C09016=1035.593,55.483,-90.705,169.074,40.767,157.648
C09017=1035.600,55.731,-90.722,169.076,40.767,157.648
C09018=1035.606,55.981,-90.739,169.078,40.766,157.648
C09019=1035.612,56.230,-90.757,169.080,40.766,157.648
C09020=1035.619,56.479,-90.774,169.082,40.766,157.648
C09021=1035.626,56.729,-90.792,169.085,40.766,157.648
C09022=1035.631,56.978,-90.809,169.087,40.765,157.648
C09023=1035.638,57.227,-90.826,169.089,40.765,157.648
C09024=1035.645,57.477,-90.844,169.091,40.764,157.648
C09025=1035.650,57.726,-90.861,169.093,40.764,157.649
C09026=1035.657,57.976,-90.878,169.095,40.764,157.649
C09027=1035.663,58.224,-90.895,169.097,40.764,157.649
C09028=1035.669,58.474,-90.913,169.100,40.763,157.649
C09029=1035.676,58.724,-90.930,169.102,40.763,157.649
C09030=1035.682,58.973,-90.948,169.104,40.762,157.649
C09031=1035.689,59.222,-90.965,169.106,40.762,157.649
C09032=1035.695,59.471,-90.983,169.108,40.762,157.649
C09033=1035.701,59.720,-91.000,169.110,40.762,157.649
C09034=1035.708,59.970,-91.017,169.113,40.761,157.649
C09035=1035.715,60.257,-91.038,169.115,40.760,157.649
C09036=1035.722,60.543,-91.058,169.117,40.760,157.649
C09037=1035.730,60.827,-91.078,169.120,40.760,157.649
C09038=1035.738,61.114,-91.098,169.122,40.760,157.649
C09039=1035.743,61.363,-91.116,169.125,40.759,157.649
C09040=1035.750,61.613,-91.133,169.127,40.759,157.649
C09041=1035.757,61.862,-91.150,169.129,40.758,157.649
C09042=1035.763,62.112,-91.168,169.131,40.758,157.649
C09043=1035.769,62.361,-91.185,169.133,40.758,157.649
C09044=1035.776,62.610,-91.203,169.135,40.758,157.649
C09045=1035.782,62.860,-91.220,169.138,40.757,157.649
C09046=1035.789,63.109,-91.238,169.140,40.756,157.649
C09047=1035.795,63.358,-91.255,169.142,40.756,157.649
C09048=1035.802,63.608,-91.273,169.144,40.756,157.649
C09049=1035.808,63.857,-91.291,169.146,40.756,157.649
C09050=1035.814,64.105,-91.308,169.148,40.755,157.650
C09051=1035.820,64.355,-91.326,169.150,40.755,157.650
C09052=1035.827,64.605,-91.344,169.152,40.755,157.650
C09053=1035.833,64.854,-91.362,169.155,40.755,157.650
C09054=1035.839,65.103,-91.380,169.157,40.754,157.650
C09055=1035.846,65.352,-91.397,169.159,40.754,157.650
C09056=1035.852,65.602,-91.415,169.161,40.754,157.650
C09057=1035.858,65.851,-91.433,169.163,40.753,157.650
C09058=1035.865,66.100,-91.451,169.165,40.753,157.650
C09059=1035.871,66.350,-91.469,169.167,40.753,157.650
C09060=1035.877,66.599,-91.487,169.169,40.752,157.650
C09061=1035.883,66.848,-91.504,169.172,40.752,157.650
C09062=1035.890,67.097,-91.522,169.174,40.752,157.650
C09063=1035.896,67.347,-91.540,169.176,40.752,157.650
C09064=1035.903,67.596,-91.557,169.178,40.751,157.650
C09065=1035.909,67.845,-91.576,169.180,40.751,157.650
C09066=1035.915,68.094,-91.594,169.182,40.751,157.650
C09067=1035.921,68.344,-91.612,169.184,40.751,157.650
C09068=1035.928,68.593,-91.630,169.186,40.751,157.650
C09069=1035.934,68.842,-91.647,169.188,40.750,157.651
C09070=1035.940,69.092,-91.665,169.192,40.750,157.651
C09071=1035.946,69.341,-91.684,169.194,40.750,157.651
C09072=1035.953,69.590,-91.701,169.196,40.750,157.651
C09073=1035.959,69.839,-91.720,169.198,40.749,157.651
C09074=1035.965,70.088,-91.737,169.200,40.749,157.651
C09075=1035.971,70.338,-91.755,169.202,40.749,157.651
C09076=1035.978,70.587,-91.774,169.204,40.749,157.651
C09077=1035.984,70.837,-91.792,169.206,40.748,157.651
C09078=1035.990,71.085,-91.810,169.208,40.748,157.651
C09079=1035.996,71.335,-91.828,169.211,40.748,157.651
C09080=1036.003,71.584,-91.846,169.213,40.748,157.651
C09081=1036.009,71.834,-91.864,169.215,40.747,157.651
C09082=1036.015,72.083,-91.883,169.217,40.747,157.651
C09083=1036.021,72.332,-91.900,169.219,40.747,157.651
C09084=1036.027,72.581,-91.919,169.221,40.747,157.651
C09085=1036.034,72.831,-91.936,169.223,40.747,157.651
C09086=1036.041,73.080,-91.955,169.225,40.746,157.652
C09087=1036.047,73.329,-91.973,169.227,40.746,157.652
C09088=1036.053,73.579,-91.992,169.229,40.746,157.652
C09089=1036.059,73.828,-92.009,169.232,40.746,157.652
C09090=1036.065,74.077,-92.028,169.234,40.745,157.652
C09091=1036.071,74.326,-92.046,169.236,40.745,157.652
C09092=1036.078,74.576,-92.064,169.238,40.745,157.652
C09093=1036.084,74.825,-92.082,169.240,40.745,157.652
C09094=1036.091,75.074,-92.100,169.242,40.744,157.652
C09095=1036.096,75.323,-92.118,169.244,40.744,157.652
C09096=1036.103,75.572,-92.137,169.246,40.744,157.652
C09097=1036.109,75.821,-92.155,169.248,40.744,157.652
C09098=1036.115,76.071,-92.173,169.251,40.743,157.652
C09099=1036.123,76.357,-92.194,169.253,40.743,157.652
C09100=1036.130,76.643,-92.215,169.255,40.743,157.652
C09101=1036.138,76.929,-92.236,169.258,40.743,157.652
C09102=1036.144,77.215,-92.257,169.260,40.742,157.653
C09103=1036.150,77.464,-92.276,169.262,40.742,157.653
C09104=1036.157,77.713,-92.294,169.264,40.742,157.653
C09105=1036.163,77.962,-92.313,169.267,40.742,157.653
C09106=1036.169,78.212,-92.331,169.269,40.741,157.653
C09107=1036.176,78.461,-92.350,169.271,40.741,157.653
C09108=1036.182,78.710,-92.368,169.273,40.741,157.653
C09109=1036.188,78.959,-92.386,169.275,40.741,157.653
C09110=1036.194,79.209,-92.404,169.278,40.741,157.653
C09111=1036.200,79.458,-92.424,169.280,40.740,157.653
C09112=1036.206,79.707,-92.442,169.282,40.740,157.653
C09113=1036.212,79.957,-92.460,169.284,40.740,157.653
C09114=1036.219,80.206,-92.479,169.286,40.740,157.653
C09115=1036.225,80.455,-92.498,169.288,40.740,157.653
C09116=1036.232,80.704,-92.516,169.290,40.740,157.653
C09117=1036.238,80.953,-92.535,169.293,40.740,157.654
C09118=1036.243,81.203,-92.553,169.295,40.739,157.654
C09119=1036.249,81.452,-92.572,169.297,40.739,157.654
C09120=1036.256,81.701,-92.590,169.299,40.739,157.654
C09121=1036.262,81.950,-92.609,169.301,40.739,157.654
C09122=1036.268,82.199,-92.628,169.303,40.738,157.654
C09123=1036.275,82.449,-92.646,169.305,40.738,157.654
C09124=1036.280,82.698,-92.665,169.307,40.738,157.654
C09125=1036.287,82.947,-92.683,169.309,40.738,157.654
C09126=1036.293,83.197,-92.702,169.311,40.738,157.654
C09127=1036.300,83.446,-92.721,169.314,40.737,157.654
C09128=1036.306,83.695,-92.739,169.316,40.737,157.654
C09129=1036.312,83.944,-92.759,169.318,40.737,157.654
C09130=1036.318,84.193,-92.777,169.320,40.737,157.654
C09131=1036.324,84.443,-92.795,169.322,40.737,157.654
C09132=1036.331,84.692,-92.814,169.324,40.737,157.655
C09133=1036.337,84.941,-92.832,169.326,40.737,157.655
C09134=1036.343,85.190,-92.851,169.328,40.736,157.655
C09135=1036.349,85.440,-92.870,169.330,40.736,157.655
C09136=1036.356,85.689,-92.889,169.332,40.736,157.655
C09137=1036.362,85.938,-92.908,169.335,40.736,157.655
C09138=1036.368,86.187,-92.926,169.338,40.735,157.655
C09139=1036.375,86.436,-92.945,169.340,40.735,157.655
C09140=1036.381,86.686,-92.964,169.342,40.735,157.655
C09141=1036.387,86.935,-92.983,169.344,40.735,157.655
C09142=1036.393,87.184,-93.001,169.346,40.734,157.655
C09143=1036.400,87.433,-93.020,169.348,40.734,157.655
C09144=1036.406,87.682,-93.039,169.350,40.734,157.655
C09145=1036.412,87.932,-93.058,169.353,40.734,157.655
C09146=1036.418,88.181,-93.077,169.355,40.733,157.655
C09147=1036.425,88.430,-93.095,169.357,40.733,157.655
C09148=1036.431,88.679,-93.114,169.359,40.733,157.655
C09149=1036.438,88.928,-93.133,169.361,40.733,157.656
C09150=1036.443,89.178,-93.152,169.363,40.733,157.656
C09151=1036.450,89.427,-93.171,169.365,40.732,157.656
C09152=1036.456,89.676,-93.189,169.367,40.732,157.656
C09153=1036.463,89.925,-93.208,169.370,40.732,157.656
C09154=1036.468,90.174,-93.227,169.372,40.732,157.656
C09155=1036.475,90.424,-93.246,169.374,40.731,157.656
C09156=1036.481,90.674,-93.265,169.376,40.732,157.656
C09157=1036.488,90.922,-93.285,169.378,40.731,157.656
C09158=1036.493,91.172,-93.304,169.380,40.731,157.656
C09159=1036.500,91.421,-93.323,169.382,40.731,157.656
C09160=1036.506,91.670,-93.341,169.384,40.731,157.656
C09161=1036.512,91.919,-93.360,169.386,40.731,157.656
C09162=1036.518,92.168,-93.379,169.388,40.730,157.656
C09163=1036.526,92.454,-93.401,169.391,40.731,157.657
C09164=1036.532,92.740,-93.423,169.393,40.730,157.657
C09165=1036.539,93.026,-93.446,169.396,40.730,157.657
C09166=1036.546,93.312,-93.467,169.399,40.730,157.657
C09167=1036.553,93.561,-93.487,169.401,40.730,157.657
C09168=1036.559,93.810,-93.506,169.403,40.729,157.657
C09169=1036.565,94.059,-93.525,169.405,40.730,157.657
C09170=1036.571,94.309,-93.544,169.407,40.730,157.657
C09171=1036.577,94.557,-93.563,169.410,40.729,157.657
C09172=1036.583,94.807,-93.582,169.412,40.729,157.657
C09173=1036.590,95.056,-93.601,169.414,40.729,157.657
C09174=1036.596,95.306,-93.621,169.416,40.729,157.657
C09175=1036.603,95.554,-93.640,169.418,40.728,157.657
C09176=1036.608,95.804,-93.659,169.420,40.728,157.657
C09177=1036.615,96.053,-93.678,169.422,40.728,157.658
C09178=1036.621,96.302,-93.698,169.424,40.728,157.658
C09179=1036.627,96.551,-93.717,169.426,40.728,157.658
C09180=1036.633,96.800,-93.736,169.429,40.728,157.658
C09181=1036.640,97.049,-93.755,169.431,40.728,157.658
C09182=1036.646,97.299,-93.775,169.433,40.727,157.658
C09183=1036.652,97.548,-93.793,169.435,40.727,157.658
C09184=1036.658,97.797,-93.813,169.437,40.727,157.658
C09185=1036.665,98.046,-93.832,169.439,40.727,157.658
C09186=1036.670,98.295,-93.851,169.441,40.727,157.658
C09187=1036.678,98.545,-93.871,169.443,40.727,157.658
C09188=1036.683,98.794,-93.890,169.447,40.727,157.658
C09189=1036.690,99.042,-93.910,169.449,40.726,157.659
C09190=1036.696,99.292,-93.929,169.451,40.726,157.659
C09191=1036.702,99.541,-93.947,169.453,40.726,157.659
C09192=1036.709,99.791,-93.968,169.455,40.726,157.659
C09193=1036.715,100.040,-93.986,169.457,40.726,157.659
C09194=1036.721,100.288,-94.006,169.459,40.725,157.659
C09195=1036.727,100.538,-94.026,169.461,40.725,157.659
C09196=1036.733,100.787,-94.046,169.464,40.725,157.659
C09197=1036.739,101.036,-94.064,169.466,40.725,157.659
C09198=1036.746,101.285,-94.085,169.468,40.725,157.659
C09199=1036.752,101.535,-94.104,169.470,40.725,157.659
C09200=1036.758,101.784,-94.124,169.472,40.725,157.659
C09201=1036.764,102.033,-94.142,169.474,40.725,157.659
C09202=1036.770,102.282,-94.162,169.476,40.725,157.660
C09203=1036.776,102.532,-94.182,169.478,40.724,157.660
C09204=1036.782,102.780,-94.202,169.480,40.724,157.660
C09205=1036.788,103.029,-94.222,169.482,40.725,157.660
C09206=1036.795,103.278,-94.241,169.485,40.724,157.660
C09207=1036.801,103.527,-94.261,169.487,40.724,157.660
C09208=1036.807,103.777,-94.280,169.489,40.724,157.660
C09209=1036.813,104.026,-94.300,169.491,40.724,157.660
C09210=1036.819,104.275,-94.320,169.494,40.724,157.660
C09211=1036.825,104.524,-94.339,169.496,40.724,157.660
C09212=1036.832,104.774,-94.359,169.498,40.724,157.660
C09213=1036.838,105.023,-94.378,169.500,40.723,157.660
C09214=1036.844,105.272,-94.398,169.503,40.723,157.660
C09215=1036.850,105.521,-94.418,169.505,40.724,157.661
C09216=1036.857,105.771,-94.437,169.507,40.723,157.661
C09217=1036.863,106.019,-94.457,169.509,40.723,157.661
C09218=1036.869,106.268,-94.477,169.511,40.723,157.661
C09219=1036.874,106.518,-94.496,169.513,40.723,157.661
C09220=1036.881,106.767,-94.517,169.515,40.723,157.661
C09221=1036.888,107.016,-94.536,169.517,40.723,157.661
C09222=1036.894,107.264,-94.556,169.520,40.723,157.661
C09223=1036.899,107.514,-94.575,169.522,40.722,157.661
C09224=1036.906,107.763,-94.596,169.524,40.722,157.661
C09225=1036.912,108.012,-94.616,169.526,40.722,157.661
C09226=1036.918,108.261,-94.634,169.529,40.722,157.662
C09227=1036.925,108.547,-94.657,169.532,40.722,157.662
C09228=1036.934,108.833,-94.681,169.534,40.722,157.662
C09229=1036.940,109.119,-94.703,169.537,40.721,157.662
C09230=1036.948,109.405,-94.726,169.539,40.721,157.662
C09231=1036.953,109.654,-94.745,169.541,40.721,157.662
C09232=1036.959,109.903,-94.765,169.543,40.721,157.662
C09233=1036.966,110.153,-94.785,169.545,40.721,157.662
C09234=1036.972,110.401,-94.805,169.548,40.721,157.662
C09235=1036.978,110.650,-94.825,169.550,40.721,157.662
C09236=1036.984,110.900,-94.845,169.552,40.720,157.662
C09237=1036.990,111.149,-94.865,169.554,40.721,157.663
C09238=1036.996,111.398,-94.885,169.556,40.721,157.663
C09239=1037.004,111.647,-94.905,169.558,40.720,157.663
C09240=1037.010,111.896,-94.924,169.560,40.720,157.663
C09241=1037.016,112.145,-94.944,169.563,40.720,157.663
C09242=1037.022,112.394,-94.965,169.565,40.720,157.663
C09243=1037.028,112.643,-94.985,169.567,40.720,157.663
C09244=1037.035,112.893,-95.005,169.569,40.720,157.663
C09245=1037.040,113.142,-95.024,169.572,40.720,157.663
C09246=1037.046,113.391,-95.044,169.574,40.720,157.663
C09247=1037.052,113.641,-95.065,169.576,40.720,157.663
C09248=1037.058,113.890,-95.085,169.579,40.720,157.664
C09249=1037.064,114.138,-95.105,169.581,40.720,157.664
C09250=1037.071,114.388,-95.125,169.583,40.720,157.664
C09251=1037.076,114.637,-95.146,169.585,40.720,157.664
C09252=1037.082,114.886,-95.166,169.587,40.720,157.664
C09253=1037.089,115.135,-95.187,169.589,40.720,157.664
C09254=1037.095,115.383,-95.207,169.591,40.720,157.664
C09255=1037.100,115.610,-95.225,169.593,40.720,157.664
C09256=1037.105,115.836,-95.243,169.595,40.720,157.664
C09257=1037.111,116.063,-95.262,169.598,40.720,157.664
C09258=1037.116,116.289,-95.280,169.600,40.720,157.665
C09259=1037.122,116.516,-95.299,169.602,40.720,157.665
C09260=1037.127,116.742,-95.318,169.604,40.720,157.665
C09261=1037.133,116.968,-95.336,169.606,40.720,157.665
C09262=1037.139,117.194,-95.354,169.608,40.719,157.665
C09263=1037.144,117.443,-95.375,169.610,40.720,157.665
C09264=1037.151,117.693,-95.395,169.612,40.720,157.665
C09265=1037.157,117.941,-95.415,169.614,40.719,157.665
C09266=1037.163,118.190,-95.435,169.616,40.720,157.665
C09267=1037.169,118.440,-95.456,169.618,40.720,157.665
C09268=1037.175,118.688,-95.477,169.621,40.720,157.666
C09269=1037.181,118.938,-95.497,169.623,40.720,157.666
C09270=1037.187,119.187,-95.517,169.625,40.720,157.666
C09271=1037.193,119.436,-95.538,169.628,40.720,157.666
C09272=1037.199,119.685,-95.558,169.630,40.720,157.666
C09273=1037.205,119.934,-95.578,169.632,40.719,157.666
C09274=1037.211,120.183,-95.600,169.635,40.720,157.666
C09275=1037.217,120.432,-95.620,169.637,40.720,157.666
C09276=1037.224,120.682,-95.640,169.639,40.719,157.666
C09277=1037.230,120.930,-95.660,169.641,40.720,157.667
C09278=1037.236,121.180,-95.682,169.643,40.720,157.667
C09279=1037.242,121.428,-95.701,169.645,40.719,157.667
C09280=1037.249,121.678,-95.722,169.648,40.720,157.667
C09281=1037.254,121.927,-95.742,169.650,40.719,157.667
C09282=1037.261,122.176,-95.763,169.652,40.719,157.667
C09283=1037.267,122.425,-95.783,169.655,40.720,157.667
C09284=1037.273,122.674,-95.804,169.657,40.719,157.667
C09285=1037.279,122.923,-95.824,169.659,40.719,157.667
C09286=1037.286,123.172,-95.845,169.662,40.719,157.667
C09287=1037.292,123.421,-95.865,169.664,40.719,157.667
C09288=1037.297,123.671,-95.886,169.666,40.719,157.668
C09289=1037.304,123.919,-95.907,169.668,40.719,157.668
C09290=1037.310,124.169,-95.927,169.670,40.719,157.668
C09291=1037.318,124.500,-95.954,169.673,40.719,157.668
C09292=1037.326,124.831,-95.982,169.676,40.719,157.668
C09293=1037.335,125.162,-96.010,169.679,40.719,157.668
C09294=1037.343,125.494,-96.037,169.682,40.719,157.668
C09295=1037.349,125.743,-96.057,169.685,40.719,157.668
C09296=1037.356,125.992,-96.078,169.687,40.719,157.668
C09297=1037.362,126.241,-96.098,169.690,40.718,157.669
C09298=1037.367,126.490,-96.119,169.692,40.719,157.669
C09299=1037.374,126.739,-96.140,169.694,40.719,157.669
C09300=1037.380,126.988,-96.160,169.696,40.718,157.669
C09301=1037.387,127.237,-96.182,169.699,40.719,157.669
C09302=1037.393,127.486,-96.202,169.701,40.718,157.669
C09303=1037.399,127.736,-96.222,169.703,40.718,157.669
C09304=1037.405,127.985,-96.244,169.705,40.719,157.669
C09305=1037.411,128.234,-96.264,169.707,40.718,157.669
C09306=1037.418,128.482,-96.285,169.710,40.718,157.669
C09307=1037.424,128.732,-96.305,169.712,40.718,157.670
C09308=1037.430,128.980,-96.326,169.714,40.718,157.670
C09309=1037.437,129.230,-96.346,169.716,40.718,157.670
C09310=1037.442,129.478,-96.368,169.720,40.718,157.670
C09311=1037.449,129.728,-96.388,169.722,40.718,157.670
C09312=1037.456,129.977,-96.409,169.724,40.718,157.670
C09313=1037.461,130.226,-96.430,169.726,40.718,157.670
C09314=1037.468,130.475,-96.451,169.729,40.717,157.670
C09315=1037.475,130.724,-96.471,169.731,40.718,157.670
C09316=1037.480,130.973,-96.492,169.733,40.718,157.670
C09317=1037.487,131.222,-96.513,169.735,40.718,157.671
C09318=1037.493,131.472,-96.534,169.737,40.718,157.671
C09319=1037.499,131.720,-96.556,169.740,40.717,157.671
C09320=1037.505,131.970,-96.576,169.742,40.718,157.671
C09321=1037.511,132.218,-96.597,169.744,40.718,157.671
C09322=1037.518,132.467,-96.618,169.747,40.718,157.671
C09323=1037.524,132.717,-96.639,169.750,40.718,157.671
C09324=1037.529,132.965,-96.660,169.752,40.718,157.671
C09325=1037.536,133.214,-96.681,169.754,40.718,157.672
C09326=1037.542,133.464,-96.702,169.756,40.718,157.672
C09327=1037.547,133.713,-96.724,169.758,40.718,157.672
C09328=1037.554,133.962,-96.745,169.761,40.718,157.672
C09329=1037.560,134.211,-96.766,169.763,40.718,157.672
C09330=1037.566,134.460,-96.787,169.765,40.718,157.672
C09331=1037.573,134.709,-96.808,169.767,40.718,157.672
C09332=1037.579,134.958,-96.830,169.770,40.718,157.672
C09333=1037.584,135.207,-96.850,169.773,40.718,157.673
C09334=1037.591,135.456,-96.871,169.775,40.718,157.673
C09335=1037.597,135.705,-96.893,169.777,40.719,157.673
C09336=1037.603,135.954,-96.914,169.779,40.718,157.673
C09337=1037.609,136.203,-96.934,169.782,40.719,157.673
C09338=1037.615,136.452,-96.956,169.784,40.718,157.673
C09339=1037.621,136.701,-96.977,169.786,40.718,157.673
C09340=1037.628,136.950,-96.998,169.788,40.719,157.673
C09341=1037.634,137.199,-97.020,169.791,40.718,157.673
C09342=1037.640,137.449,-97.041,169.793,40.719,157.674
C09343=1037.645,137.697,-97.062,169.795,40.719,157.674
C09344=1037.652,137.946,-97.083,169.798,40.719,157.674
C09345=1037.659,138.195,-97.105,169.801,40.719,157.674
C09346=1037.664,138.444,-97.126,169.803,40.719,157.674
C09347=1037.671,138.693,-97.147,169.805,40.719,157.674
C09348=1037.677,138.942,-97.169,169.807,40.719,157.674
C09349=1037.683,139.191,-97.190,169.810,40.719,157.674
C09350=1037.689,139.440,-97.211,169.812,40.719,157.675
C09351=1037.695,139.690,-97.233,169.814,40.719,157.675
C09352=1037.701,139.939,-97.254,169.817,40.719,157.675
C09353=1037.707,140.188,-97.276,169.820,40.719,157.675
C09354=1037.713,140.436,-97.296,169.822,40.720,157.675
C09355=1037.721,140.722,-97.322,169.825,40.720,157.675
C09356=1037.727,141.007,-97.347,169.827,40.720,157.675
C09357=1037.735,141.293,-97.371,169.830,40.720,157.676
C09358=1037.741,141.578,-97.396,169.832,40.720,157.676
C09359=1037.747,141.827,-97.417,169.835,40.720,157.676
C09360=1037.753,142.076,-97.439,169.838,40.720,157.676
C09361=1037.759,142.325,-97.460,169.840,40.720,157.676
C09362=1037.765,142.574,-97.482,169.842,40.721,157.676
C09363=1037.772,142.824,-97.504,169.845,40.720,157.676
C09364=1037.778,143.073,-97.525,169.847,40.721,157.677
C09365=1037.784,143.321,-97.546,169.849,40.720,157.677
C09366=1037.790,143.570,-97.568,169.851,40.721,157.677
C09367=1037.796,143.819,-97.589,169.854,40.721,157.677
C09368=1037.802,144.069,-97.611,169.856,40.721,157.677
C09369=1037.809,144.317,-97.633,169.859,40.721,157.677
C09370=1037.814,144.566,-97.654,169.862,40.721,157.677
C09371=1037.821,144.815,-97.676,169.864,40.721,157.678
C09372=1037.827,145.064,-97.698,169.866,40.721,157.678
C09373=1037.833,145.313,-97.719,169.868,40.722,157.678
C09374=1037.839,145.563,-97.741,169.871,40.721,157.678
C09375=1037.845,145.812,-97.763,169.873,40.722,157.678
C09376=1037.851,146.060,-97.785,169.875,40.721,157.678
C09377=1037.857,146.309,-97.806,169.878,40.722,157.678
C09378=1037.864,146.558,-97.828,169.881,40.722,157.679
C09379=1037.870,146.807,-97.849,169.883,40.722,157.679
C09380=1037.876,147.056,-97.871,169.886,40.722,157.679
C09381=1037.882,147.305,-97.893,169.888,40.722,157.679
C09382=1037.888,147.554,-97.915,169.890,40.722,157.679
C09383=1037.895,147.803,-97.937,169.892,40.723,157.679
C09384=1037.900,148.052,-97.958,169.895,40.723,157.679
C09385=1037.907,148.300,-97.980,169.897,40.723,157.679
C09386=1037.913,148.550,-98.002,169.899,40.723,157.680
C09387=1037.919,148.799,-98.024,169.903,40.723,157.680
C09388=1037.925,149.048,-98.045,169.905,40.723,157.680
C09389=1037.931,149.297,-98.068,169.907,40.723,157.680
C09390=1037.937,149.546,-98.090,169.910,40.724,157.680
C09391=1037.943,149.795,-98.111,169.912,40.724,157.680
C09392=1037.949,150.043,-98.133,169.914,40.724,157.680
C09393=1037.955,150.293,-98.155,169.916,40.724,157.681
C09394=1037.962,150.541,-98.177,169.919,40.724,157.681
C09395=1037.967,150.791,-98.200,169.922,40.725,157.681
C09396=1037.973,151.040,-98.221,169.924,40.725,157.681
C09397=1037.980,151.288,-98.244,169.927,40.725,157.681
C09398=1037.986,151.538,-98.265,169.929,40.725,157.681
C09399=1037.992,151.786,-98.288,169.931,40.725,157.682
C09400=1037.998,152.036,-98.310,169.934,40.725,157.682
C09401=1038.004,152.285,-98.332,169.936,40.726,157.682
C09402=1038.010,152.534,-98.354,169.938,40.726,157.682
C09403=1038.017,152.783,-98.376,169.942,40.726,157.682
C09404=1038.022,153.031,-98.398,169.944,40.726,157.682
C09405=1038.028,153.280,-98.420,169.946,40.726,157.682
C09406=1038.034,153.529,-98.442,169.949,40.726,157.683
C09407=1038.041,153.778,-98.464,169.951,40.727,157.683
C09408=1038.047,154.026,-98.486,169.953,40.727,157.683
C09409=1038.053,154.276,-98.508,169.956,40.727,157.683
C09410=1038.059,154.525,-98.531,169.959,40.727,157.683
C09411=1038.065,154.774,-98.552,169.961,40.728,157.683
C09412=1038.072,155.022,-98.575,169.964,40.727,157.684
C09413=1038.077,155.272,-98.597,169.966,40.728,157.684
C09414=1038.083,155.520,-98.619,169.968,40.728,157.684
C09415=1038.090,155.769,-98.642,169.971,40.728,157.684
C09416=1038.095,156.019,-98.664,169.973,40.728,157.684
C09417=1038.102,156.267,-98.686,169.977,40.729,157.684
C09418=1038.108,156.516,-98.708,169.979,40.729,157.685
C09419=1038.115,156.802,-98.734,169.982,40.729,157.685
C09420=1038.121,157.087,-98.759,169.984,40.729,157.685
C09421=1038.129,157.372,-98.785,169.987,40.729,157.685
C09422=1038.135,157.657,-98.810,169.990,40.730,157.685
C09423=1038.142,157.906,-98.833,169.993,40.730,157.685
C09424=1038.148,158.154,-98.855,169.995,40.730,157.686
C09425=1038.154,158.404,-98.877,169.998,40.730,157.686
C09426=1038.160,158.652,-98.900,170.000,40.731,157.686
C09427=1038.166,158.901,-98.923,170.003,40.731,157.686
C09428=1038.172,159.150,-98.945,170.005,40.731,157.686
C09429=1038.179,159.400,-98.967,170.007,40.732,157.686
C09430=1038.185,159.649,-98.990,170.011,40.731,157.687
C09431=1038.191,159.897,-99.012,170.013,40.732,157.687
C09432=1038.197,160.146,-99.035,170.015,40.732,157.687
C09433=1038.203,160.395,-99.057,170.018,40.732,157.687
C09434=1038.209,160.644,-99.080,170.020,40.733,157.687
C09435=1038.215,160.893,-99.103,170.022,40.733,157.688
C09436=1038.220,161.142,-99.126,170.026,40.734,157.688
C09437=1038.227,161.391,-99.148,170.028,40.734,157.688
C09438=1038.233,161.640,-99.171,170.031,40.734,157.688
C09439=1038.238,161.888,-99.194,170.033,40.735,157.688
C09440=1038.244,162.137,-99.217,170.035,40.735,157.689
C09441=1038.250,162.386,-99.240,170.039,40.735,157.689
C09442=1038.256,162.635,-99.261,170.041,40.736,157.689
C09443=1038.262,162.884,-99.284,170.043,40.736,157.689
C09444=1038.267,163.133,-99.307,170.046,40.736,157.689
C09445=1038.273,163.382,-99.330,170.048,40.737,157.690
C09446=1038.280,163.631,-99.353,170.050,40.737,157.690
C09447=1038.285,163.880,-99.376,170.054,40.738,157.690
C09448=1038.291,164.129,-99.399,170.056,40.738,157.690
C09449=1038.297,164.377,-99.422,170.059,40.738,157.690
C09450=1038.303,164.626,-99.444,170.061,40.739,157.690
C09451=1038.310,164.876,-99.467,170.063,40.739,157.691
C09452=1038.315,165.125,-99.490,170.067,40.739,157.691
C09453=1038.321,165.373,-99.513,170.069,40.740,157.691
C09454=1038.327,165.622,-99.536,170.071,40.740,157.691
C09455=1038.333,165.871,-99.560,170.074,40.741,157.691
C09456=1038.339,166.119,-99.582,170.076,40.741,157.692
C09457=1038.345,166.368,-99.605,170.079,40.741,157.692
C09458=1038.351,166.617,-99.628,170.082,40.742,157.692
C09459=1038.357,166.866,-99.651,170.084,40.742,157.692
C09460=1038.363,167.115,-99.674,170.087,40.742,157.692
C09461=1038.369,167.364,-99.697,170.089,40.743,157.693
C09462=1038.375,167.613,-99.719,170.092,40.743,157.693
C09463=1038.381,167.862,-99.742,170.095,40.743,157.693
C09464=1038.387,168.110,-99.766,170.098,40.744,157.693
C09465=1038.393,168.359,-99.789,170.100,40.744,157.693
C09466=1038.400,168.608,-99.812,170.102,40.745,157.694
C09467=1038.405,168.857,-99.835,170.105,40.745,157.694
C09468=1038.411,169.106,-99.858,170.107,40.745,157.694
C09469=1038.417,169.355,-99.881,170.111,40.746,157.694
C09470=1038.423,169.603,-99.904,170.113,40.746,157.694
C09471=1038.429,169.853,-99.928,170.116,40.746,157.695
C09472=1038.436,170.101,-99.950,170.118,40.747,157.695
C09473=1038.441,170.350,-99.973,170.121,40.747,157.695
C09474=1038.447,170.599,-99.996,170.124,40.747,157.695
C09475=1038.453,170.848,-100.019,170.126,40.748,157.695
C09476=1038.459,171.097,-100.043,170.129,40.748,157.696
C09477=1038.465,171.346,-100.066,170.131,40.748,157.696
C09478=1038.472,171.595,-100.088,170.134,40.749,157.696
C09479=1038.478,171.843,-100.112,170.136,40.749,157.696
C09480=1038.484,172.093,-100.135,170.140,40.749,157.696
C09481=1038.490,172.341,-100.158,170.142,40.750,157.697
C09482=1038.496,172.590,-100.182,170.145,40.750,157.697
C09483=1038.503,172.875,-100.208,170.148,40.750,157.697
C09484=1038.510,173.159,-100.235,170.150,40.751,157.697
C09485=1038.517,173.444,-100.261,170.154,40.751,157.697
C09486=1038.524,173.729,-100.288,170.157,40.752,157.698
C09487=1038.530,173.978,-100.311,170.160,40.752,157.698
C09488=1038.536,174.226,-100.333,170.162,40.753,157.698
C09489=1038.543,174.475,-100.357,170.166,40.753,157.698
C09490=1038.549,174.724,-100.380,170.168,40.753,157.699
C09491=1038.555,174.973,-100.404,170.171,40.754,157.699
C09492=1038.561,175.222,-100.427,170.173,40.754,157.699
C09493=1038.567,175.471,-100.450,170.176,40.754,157.699
C09494=1038.573,175.719,-100.474,170.178,40.755,157.699
C09495=1038.579,175.968,-100.496,170.182,40.755,157.700
C09496=1038.586,176.217,-100.520,170.184,40.756,157.700
C09497=1038.592,176.466,-100.543,170.187,40.756,157.700
C09498=1038.598,176.715,-100.567,170.189,40.756,157.700
C09499=1038.604,176.964,-100.590,170.192,40.757,157.700
C09500=1038.610,177.212,-100.614,170.195,40.757,157.701
C09501=1038.617,177.462,-100.637,170.198,40.757,157.701
C09502=1038.623,177.710,-100.661,170.200,40.758,157.701
C09503=1038.630,177.959,-100.684,170.203,40.758,157.701
C09504=1038.636,178.207,-100.707,170.206,40.758,157.701
C09505=1038.641,178.456,-100.730,170.209,40.759,157.702
C09506=1038.648,178.705,-100.754,170.212,40.760,157.702
C09507=1038.654,178.954,-100.777,170.214,40.760,157.702
C09508=1038.660,179.203,-100.801,170.217,40.760,157.702
C09509=1038.666,179.452,-100.824,170.219,40.761,157.703
C09510=1038.673,179.701,-100.848,170.223,40.761,157.703
C09511=1038.679,179.950,-100.871,170.225,40.761,157.703
C09512=1038.685,180.198,-100.894,170.228,40.762,157.703
C09513=1038.692,180.447,-100.918,170.231,40.762,157.703
C09514=1038.698,180.696,-100.941,170.233,40.762,157.704
C09515=1038.704,180.945,-100.965,170.236,40.763,157.704
C09516=1038.710,181.193,-100.989,170.239,40.763,157.704
C09517=1038.717,181.443,-101.012,170.242,40.764,157.704
C09518=1038.723,181.691,-101.036,170.245,40.764,157.705
C09519=1038.729,181.940,-101.060,170.247,40.765,157.705
C09520=1038.735,182.189,-101.083,170.251,40.765,157.705
C09521=1038.742,182.438,-101.107,170.253,40.765,157.705
C09522=1038.748,182.686,-101.130,170.256,40.766,157.705
C09523=1038.755,182.935,-101.153,170.259,40.766,157.706
C09524=1038.761,183.184,-101.177,170.261,40.766,157.706
C09525=1038.768,183.433,-101.201,170.265,40.767,157.706
C09526=1038.773,183.682,-101.225,170.267,40.768,157.706
C09527=1038.779,183.930,-101.249,170.270,40.768,157.706
C09528=1038.784,184.179,-101.273,170.272,40.769,157.707
C09529=1038.791,184.428,-101.297,170.276,40.769,157.707
C09530=1038.796,184.677,-101.321,170.279,40.770,157.707
C09531=1038.803,184.926,-101.345,170.281,40.771,157.708
C09532=1038.809,185.174,-101.369,170.284,40.771,157.708
C09533=1038.815,185.423,-101.393,170.287,40.772,157.708
C09534=1038.821,185.672,-101.417,170.290,40.772,157.708
C09535=1038.826,185.920,-101.441,170.292,40.773,157.709
C09536=1038.833,186.169,-101.465,170.295,40.774,157.709
C09537=1038.838,186.418,-101.489,170.298,40.774,157.709
C09538=1038.845,186.667,-101.514,170.301,40.775,157.709
C09539=1038.850,186.915,-101.538,170.304,40.775,157.710
C09540=1038.857,187.164,-101.562,170.306,40.776,157.710
C09541=1038.862,187.413,-101.586,170.310,40.776,157.710
C09542=1038.869,187.662,-101.610,170.312,40.777,157.710
C09543=1038.874,187.911,-101.634,170.315,40.778,157.711
C09544=1038.881,188.160,-101.658,170.318,40.778,157.711
C09545=1038.887,188.409,-101.683,170.321,40.779,157.711
C09546=1038.893,188.657,-101.707,170.324,40.779,157.711
C09547=1038.900,188.941,-101.735,170.327,40.780,157.712
C09548=1038.907,189.225,-101.762,170.331,40.781,157.712
C09549=1038.913,189.510,-101.790,170.334,40.781,157.712
C09550=1038.920,189.794,-101.818,170.337,40.782,157.713
C09551=1038.926,190.043,-101.842,170.339,40.783,157.713
C09552=1038.932,190.292,-101.867,170.343,40.784,157.713
C09553=1038.938,190.540,-101.890,170.346,40.785,157.714
C09554=1038.944,190.789,-101.915,170.348,40.785,157.714
C09555=1038.951,191.038,-101.940,170.352,40.786,157.714
C09556=1038.957,191.286,-101.964,170.354,40.786,157.714
C09557=1038.963,191.535,-101.988,170.357,40.787,157.715
C09558=1038.968,191.784,-102.012,170.360,40.788,157.715
C09559=1038.975,192.033,-102.036,170.362,40.788,157.715
C09560=1038.981,192.282,-102.062,170.366,40.789,157.715
C09561=1038.987,192.530,-102.085,170.369,40.789,157.716
C09562=1038.993,192.779,-102.110,170.371,40.790,157.716
C09563=1039.000,193.027,-102.135,170.374,40.790,157.716
C09564=1039.005,193.276,-102.159,170.378,40.791,157.717
C09565=1039.011,193.525,-102.184,170.380,40.792,157.717
C09566=1039.018,193.774,-102.208,170.383,40.793,157.717
C09567=1039.024,194.022,-102.233,170.387,40.794,157.717
C09568=1039.030,194.271,-102.257,170.389,40.794,157.718
C09569=1039.036,194.521,-102.281,170.392,40.795,157.718
C09570=1039.043,194.768,-102.306,170.395,40.795,157.718
C09571=1039.048,195.018,-102.330,170.398,40.796,157.718
C09572=1039.055,195.267,-102.354,170.401,40.797,157.719
C09573=1039.061,195.515,-102.380,170.404,40.797,157.719
C09574=1039.067,195.763,-102.403,170.408,40.798,157.719
C09575=1039.074,196.012,-102.429,170.410,40.799,157.720
C09576=1039.080,196.261,-102.453,170.413,40.799,157.720
C09577=1039.086,196.510,-102.477,170.416,40.800,157.720
C09578=1039.092,196.758,-102.502,170.419,40.801,157.720
C09579=1039.098,197.007,-102.526,170.422,40.801,157.721
C09580=1039.104,197.256,-102.552,170.425,40.802,157.721
C09581=1039.111,197.505,-102.576,170.428,40.802,157.721
C09582=1039.117,197.753,-102.601,170.431,40.803,157.722
C09583=1039.123,198.002,-102.625,170.434,40.804,157.722
C09584=1039.130,198.251,-102.650,170.437,40.805,157.722
C09585=1039.136,198.500,-102.674,170.440,40.806,157.722
C09586=1039.142,198.748,-102.699,170.443,40.806,157.723
C09587=1039.148,198.997,-102.724,170.446,40.807,157.723
C09588=1039.155,199.245,-102.748,170.449,40.807,157.723
C09589=1039.161,199.494,-102.773,170.452,40.808,157.724
C09590=1039.168,199.743,-102.798,170.455,40.809,157.724
C09591=1039.173,199.992,-102.822,170.458,40.809,157.724
C09592=1039.180,200.240,-102.847,170.462,40.810,157.724
C09593=1039.186,200.488,-102.872,170.465,40.811,157.725
C09594=1039.192,200.738,-102.897,170.467,40.812,157.725
C09595=1039.199,200.986,-102.921,170.471,40.813,157.725
C09596=1039.205,201.235,-102.947,170.474,40.813,157.726
C09597=1039.211,201.484,-102.971,170.477,40.814,157.726
C09598=1039.217,201.733,-102.997,170.479,40.815,157.726
C09599=1039.223,201.981,-103.022,170.483,40.816,157.727
C09600=1039.229,202.229,-103.047,170.486,40.817,157.727
C09601=1039.235,202.479,-103.072,170.490,40.817,157.727
C09602=1039.241,202.727,-103.097,170.492,40.818,157.727
C09603=1039.247,202.976,-103.122,170.495,40.819,157.728
C09604=1039.254,203.224,-103.147,170.498,40.820,157.728
C09605=1039.260,203.474,-103.172,170.502,40.821,157.729
C09606=1039.266,203.722,-103.197,170.504,40.822,157.729
C09607=1039.272,203.970,-103.222,170.507,40.822,157.729
C09608=1039.278,204.219,-103.247,170.511,40.823,157.729
C09609=1039.284,204.468,-103.273,170.514,40.824,157.730
C09610=1039.291,204.716,-103.298,170.516,40.825,157.730
C09611=1039.317,205.767,-103.405,170.811,40.929,157.766
C09612=1039.325,206.078,-103.437,170.813,40.930,157.767
C09613=1039.333,206.389,-103.470,170.816,40.933,157.767
C09614=1039.342,206.699,-103.503,170.819,40.934,157.768
C09615=1039.351,207.010,-103.535,170.822,40.936,157.769
C09616=1039.357,207.258,-103.563,170.824,40.938,157.769
C09617=1039.364,207.507,-103.589,170.826,40.939,157.769
C09618=1039.371,207.755,-103.615,170.829,40.941,157.770
C09619=1039.377,208.004,-103.642,170.831,40.942,157.770
C09620=1039.384,208.253,-103.669,170.833,40.944,157.771
C09621=1039.391,208.501,-103.695,170.835,40.946,157.771
C09622=1039.398,208.749,-103.721,170.838,40.947,157.772
C09623=1039.403,208.998,-103.748,170.840,40.949,157.772
C09624=1039.411,209.247,-103.774,170.842,40.951,157.773
C09625=1039.418,209.495,-103.801,170.844,40.952,157.773
C09626=1039.424,209.743,-103.828,170.847,40.953,157.773
C09627=1039.431,209.992,-103.854,170.849,40.955,157.774
C09628=1039.437,210.240,-103.881,170.852,40.957,157.774
C09629=1039.444,210.489,-103.908,170.853,40.958,157.775
C09630=1039.451,210.738,-103.934,170.856,40.960,157.775
C09631=1039.457,210.986,-103.961,170.858,40.962,157.776
C09632=1039.464,211.234,-103.988,170.861,40.963,157.776
C09633=1039.471,211.483,-104.014,170.863,40.965,157.777
C09634=1039.477,211.731,-104.041,170.865,40.967,157.777
C09635=1039.484,211.980,-104.067,170.867,40.968,157.777
C09636=1039.491,212.228,-104.095,170.870,40.970,157.778
C09637=1039.497,212.477,-104.122,170.872,40.971,157.778
C09638=1039.504,212.726,-104.148,170.875,40.973,157.779
C09639=1039.510,212.974,-104.176,170.876,40.974,157.779
C09640=1039.517,213.222,-104.202,170.879,40.976,157.780
C09641=1039.523,213.471,-104.229,170.881,40.978,157.780
C09642=1039.531,213.719,-104.256,170.884,40.979,157.781
C09643=1039.536,213.968,-104.283,170.886,40.981,157.781
C09644=1039.543,214.216,-104.309,170.889,40.982,157.782
C09645=1039.550,214.465,-104.337,170.890,40.984,157.782
C09646=1039.557,214.713,-104.363,170.893,40.986,157.782
C09647=1039.563,214.962,-104.390,170.895,40.987,157.783
C09648=1039.570,215.210,-104.418,170.898,40.989,157.783
C09649=1039.576,215.458,-104.444,170.900,40.991,157.784
C09650=1039.583,215.707,-104.471,170.903,40.992,157.784
C09651=1039.590,215.956,-104.498,170.904,40.993,157.785
C09652=1039.597,216.204,-104.526,170.907,40.995,157.785
C09653=1039.603,216.452,-104.552,170.909,40.997,157.786
C09654=1039.610,216.701,-104.579,170.912,40.998,157.786
C09655=1039.617,216.949,-104.606,170.914,41.000,157.787
C09656=1039.623,217.198,-104.633,170.917,41.002,157.787
C09657=1039.629,217.446,-104.660,170.919,41.003,157.787
C09658=1039.637,217.695,-104.687,170.922,41.005,157.788
C09659=1039.643,217.943,-104.714,170.923,41.006,157.788
C09660=1039.650,218.192,-104.741,170.926,41.008,157.789
C09661=1039.656,218.440,-104.768,170.928,41.009,157.789
C09662=1039.664,218.689,-104.794,170.931,41.011,157.790
C09663=1039.670,218.937,-104.822,170.933,41.012,157.790
C09664=1039.677,219.186,-104.849,170.936,41.014,157.791
C09665=1039.684,219.434,-104.876,170.938,41.016,157.791
C09666=1039.690,219.682,-104.904,170.941,41.017,157.792
C09667=1039.697,219.931,-104.930,170.943,41.019,157.792
C09668=1039.705,220.247,-104.965,170.946,41.021,157.793
C09669=1039.714,220.563,-105.000,170.948,41.023,157.793
C09670=1039.723,220.880,-105.035,170.952,41.025,157.794
C09671=1039.730,221.196,-105.069,170.955,41.027,157.794
C09672=1039.737,221.444,-105.097,170.957,41.029,157.795
C09673=1039.744,221.692,-105.124,170.960,41.030,157.795
C09674=1039.751,221.941,-105.151,170.962,41.032,157.796
C09675=1039.757,222.190,-105.179,170.965,41.034,157.796
C09676=1039.763,222.437,-105.206,170.967,41.035,157.797
C09677=1039.770,222.686,-105.234,170.970,41.037,157.797
C09678=1039.776,222.935,-105.261,170.973,41.038,157.798
C09679=1039.784,223.183,-105.288,170.975,41.040,157.798
C09680=1039.790,223.431,-105.316,170.978,41.042,157.799
C09681=1039.797,223.680,-105.344,170.979,41.043,157.799
C09682=1039.803,223.928,-105.370,170.982,41.045,157.800
C09683=1039.810,224.177,-105.398,170.984,41.047,157.800
C09684=1039.816,224.425,-105.426,170.987,41.048,157.800
C09685=1039.824,224.673,-105.453,170.989,41.050,157.801
C09686=1039.830,224.922,-105.481,170.992,41.051,157.801
C09687=1039.837,225.170,-105.508,170.994,41.052,157.802
C09688=1039.843,225.419,-105.535,170.997,41.054,157.802
C09689=1039.850,225.668,-105.563,170.999,41.056,157.803
C09690=1039.856,225.915,-105.590,171.002,41.057,157.803
C09691=1039.863,226.164,-105.618,171.004,41.059,157.804
C09692=1039.870,226.412,-105.646,171.007,41.060,157.804
C09693=1039.877,226.660,-105.673,171.009,41.062,157.805
C09694=1039.884,226.909,-105.701,171.012,41.064,157.805
C09695=1039.890,227.157,-105.729,171.014,41.065,157.806
C09696=1039.897,227.406,-105.756,171.017,41.067,157.806
C09697=1039.903,227.655,-105.783,171.019,41.069,157.806
C09698=1039.910,227.903,-105.811,171.022,41.070,157.807
C09699=1039.917,228.152,-105.839,171.024,41.072,157.807
C09700=1039.923,228.400,-105.866,171.027,41.073,157.808
C09701=1039.930,228.649,-105.894,171.029,41.075,157.808
C09702=1039.937,228.897,-105.922,171.032,41.077,157.809
C09703=1039.943,229.145,-105.950,171.034,41.078,157.809
C09704=1039.950,229.393,-105.977,171.037,41.080,157.810
C09705=1039.957,229.641,-106.005,171.039,41.081,157.810
C09706=1039.963,229.889,-106.033,171.042,41.083,157.811
C09707=1039.970,230.138,-106.061,171.045,41.085,157.811
C09708=1039.977,230.386,-106.089,171.047,41.086,157.812
C09709=1039.983,230.635,-106.116,171.050,41.088,157.812
C09710=1039.990,230.883,-106.144,171.052,41.089,157.813
C09711=1039.996,231.132,-106.172,171.055,41.091,157.813
C09712=1040.003,231.380,-106.200,171.057,41.093,157.814
C09713=1040.010,231.628,-106.229,171.060,41.094,157.814
C09714=1040.016,231.877,-106.256,171.062,41.096,157.814
C09715=1040.023,232.125,-106.284,171.065,41.097,157.815
C09716=1040.030,232.374,-106.312,171.067,41.099,157.815
C09717=1040.036,232.622,-106.340,171.070,41.101,157.816
C09718=1040.043,232.870,-106.369,171.072,41.102,157.816
C09719=1040.049,233.119,-106.396,171.075,41.104,157.817
C09720=1040.056,233.367,-106.424,171.077,41.106,157.817
C09721=1040.062,233.616,-106.452,171.080,41.107,157.818
C09722=1040.069,233.864,-106.481,171.084,41.109,157.818
C09723=1040.075,234.112,-106.509,171.086,41.111,157.819
C09724=1040.084,234.420,-106.543,171.089,41.112,157.819
C09725=1040.092,234.729,-106.579,171.092,41.115,157.820
C09726=1040.099,235.038,-106.613,171.095,41.117,157.821
C09727=1040.108,235.347,-106.648,171.099,41.119,157.821
C09728=1040.115,235.595,-106.677,171.101,41.120,157.822
C09729=1040.122,235.843,-106.705,171.104,41.122,157.822
C09730=1040.128,236.092,-106.733,171.106,41.124,157.823
C09731=1040.135,236.340,-106.761,171.109,41.125,157.823
C09732=1040.141,236.588,-106.789,171.111,41.127,157.824
C09733=1040.148,236.837,-106.817,171.114,41.128,157.824
C09734=1040.154,237.085,-106.846,171.116,41.130,157.825
C09735=1040.162,237.334,-106.874,171.120,41.132,157.825
C09736=1040.169,237.582,-106.902,171.123,41.133,157.826
C09737=1040.175,237.831,-106.931,171.125,41.135,157.826
C09738=1040.182,238.079,-106.959,171.128,41.136,157.827
C09739=1040.188,238.327,-106.987,171.130,41.138,157.827
C09740=1040.195,238.575,-107.016,171.133,41.140,157.828
C09741=1040.201,238.824,-107.044,171.135,41.142,157.828
C09742=1040.208,239.071,-107.072,171.138,41.143,157.829
C09743=1040.214,239.320,-107.100,171.140,41.145,157.829
C09744=1040.222,239.569,-107.129,171.144,41.146,157.830
C09745=1040.228,239.817,-107.157,171.146,41.148,157.830
C09746=1040.235,240.065,-107.186,171.149,41.150,157.831
C09747=1040.241,240.314,-107.214,171.152,41.151,157.831
C09748=1040.248,240.562,-107.242,171.154,41.153,157.831
C09749=1040.254,240.810,-107.270,171.157,41.154,157.832
C09750=1040.262,241.059,-107.299,171.159,41.156,157.832
C09751=1040.268,241.307,-107.328,171.163,41.158,157.833
C09752=1040.275,241.555,-107.356,171.165,41.160,157.834
C09753=1040.281,241.803,-107.385,171.168,41.161,157.834
C09754=1040.288,242.051,-107.414,171.170,41.163,157.835
C09755=1040.294,242.299,-107.443,171.173,41.165,157.835
C09756=1040.301,242.548,-107.470,171.175,41.166,157.835
C09757=1040.308,242.797,-107.500,171.178,41.168,157.836
C09758=1040.314,243.045,-107.529,171.182,41.170,157.837
C09759=1040.321,243.293,-107.557,171.184,41.171,157.837
C09760=1040.327,243.541,-107.586,171.187,41.173,157.838
C09761=1040.334,243.789,-107.614,171.189,41.175,157.838
C09762=1040.340,244.037,-107.643,171.192,41.176,157.838
C09763=1040.347,244.286,-107.672,171.194,41.178,157.839
C09764=1040.354,244.535,-107.700,171.198,41.180,157.840
C09765=1040.360,244.783,-107.729,171.201,41.181,157.840
C09766=1040.367,245.031,-107.758,171.203,41.183,157.841
C09767=1040.374,245.279,-107.787,171.206,41.185,157.841
C09768=1040.380,245.528,-107.816,171.208,41.186,157.842
C09769=1040.386,245.776,-107.845,171.212,41.188,157.842
C09770=1040.393,246.024,-107.874,171.214,41.190,157.843
C09771=1040.400,246.272,-107.903,171.217,41.192,157.843
C09772=1040.406,246.520,-107.932,171.220,41.193,157.844
C09773=1040.413,246.769,-107.961,171.222,41.195,157.844
C09774=1040.419,247.017,-107.990,171.225,41.197,157.845
C09775=1040.425,247.265,-108.019,171.228,41.198,157.845
C09776=1040.431,247.513,-108.048,171.231,41.201,157.846
C09777=1040.438,247.762,-108.078,171.234,41.202,157.846
C09778=1040.445,248.010,-108.106,171.236,41.204,157.847
C09779=1040.452,248.258,-108.135,171.239,41.205,157.847
C09780=1040.459,248.561,-108.170,171.242,41.207,157.848
C09781=1040.467,248.864,-108.206,171.246,41.210,157.849
C09782=1040.475,249.167,-108.242,171.250,41.212,157.849
C09783=1040.483,249.470,-108.277,171.252,41.214,157.850
C09784=1040.489,249.718,-108.307,171.255,41.216,157.850
C09785=1040.496,249.966,-108.336,171.259,41.218,157.851
C09786=1040.503,250.214,-108.364,171.261,41.219,157.851
C09787=1040.510,250.463,-108.393,171.264,41.221,157.852
C09788=1040.516,250.711,-108.422,171.266,41.223,157.853
C09789=1040.522,250.959,-108.452,171.270,41.224,157.853
C09790=1040.529,251.207,-108.482,171.273,41.226,157.854
C09791=1040.535,251.456,-108.511,171.275,41.228,157.854
C09792=1040.542,251.704,-108.540,171.278,41.230,157.855
C09793=1040.549,251.952,-108.569,171.281,41.231,157.855
C09794=1040.556,252.200,-108.598,171.284,41.233,157.856
C09795=1040.562,252.448,-108.627,171.287,41.235,157.856
C09796=1040.569,252.697,-108.657,171.290,41.236,157.857
C09797=1040.575,252.945,-108.686,171.293,41.238,157.857
C09798=1040.582,253.193,-108.716,171.295,41.240,157.858
C09799=1040.589,253.441,-108.745,171.298,41.242,157.858
C09800=1040.595,253.689,-108.774,171.301,41.243,157.859
C09801=1040.602,253.938,-108.803,171.304,41.245,157.859
C09802=1040.608,254.186,-108.833,171.307,41.246,157.860
C09803=1040.616,254.434,-108.862,171.310,41.249,157.860
C09804=1040.622,254.682,-108.891,171.313,41.250,157.861
C09805=1040.629,254.930,-108.921,171.315,41.252,157.861
C09806=1040.636,255.179,-108.950,171.319,41.254,157.862
C09807=1040.642,255.427,-108.979,171.322,41.255,157.863
C09808=1040.649,255.675,-109.009,171.324,41.257,157.863
C09809=1040.655,255.923,-109.038,171.328,41.258,157.864
C09810=1040.662,256.172,-109.068,171.330,41.261,157.864
C09811=1040.669,256.419,-109.097,171.333,41.262,157.865
C09812=1040.675,256.668,-109.127,171.336,41.264,157.865
C09813=1040.682,256.916,-109.157,171.339,41.265,157.866
C09814=1040.689,257.164,-109.185,171.342,41.267,157.866
C09815=1040.696,257.412,-109.215,171.345,41.269,157.867
C09816=1040.702,257.660,-109.244,171.348,41.270,157.867
C09817=1040.710,257.908,-109.274,171.351,41.273,157.868
C09818=1040.716,258.156,-109.303,171.354,41.274,157.868
C09819=1040.723,258.404,-109.334,171.357,41.276,157.869
C09820=1040.730,258.653,-109.363,171.359,41.277,157.869
C09821=1040.736,258.901,-109.393,171.363,41.279,157.870
C09822=1040.743,259.150,-109.422,171.365,41.281,157.870
C09823=1040.750,259.397,-109.452,171.369,41.282,157.871
C09824=1040.757,259.646,-109.481,171.372,41.285,157.872
C09825=1040.763,259.894,-109.511,171.374,41.286,157.872
C09826=1040.770,260.142,-109.540,171.378,41.288,157.873
C09827=1040.777,260.390,-109.570,171.380,41.289,157.873
C09828=1040.784,260.638,-109.600,171.384,41.291,157.874
C09829=1040.791,260.887,-109.629,171.387,41.293,157.874
C09830=1040.798,261.134,-109.659,171.389,41.294,157.875
C09831=1040.805,261.383,-109.688,171.393,41.296,157.875
C09832=1040.811,261.630,-109.718,171.395,41.298,157.876
C09833=1040.818,261.879,-109.748,171.399,41.299,157.876
C09834=1040.825,262.127,-109.778,171.402,41.302,157.877
C09835=1040.831,262.375,-109.808,171.405,41.303,157.877
C09836=1040.839,262.677,-109.845,171.408,41.305,157.878
C09837=1040.848,262.978,-109.881,171.412,41.307,157.879
C09838=1040.856,263.279,-109.917,171.416,41.310,157.880
C09839=1040.864,263.581,-109.954,171.419,41.312,157.880
C09840=1040.870,263.829,-109.984,171.423,41.314,157.881
C09841=1040.877,264.077,-110.013,171.426,41.316,157.881
C09842=1040.884,264.326,-110.044,171.428,41.317,157.882
C09843=1040.890,264.574,-110.074,171.432,41.319,157.882
C09844=1040.897,264.822,-110.104,171.434,41.321,157.883
C09845=1040.904,265.070,-110.134,171.438,41.323,157.884
C09846=1040.910,265.318,-110.164,171.441,41.325,157.884
C09847=1040.917,265.566,-110.195,171.444,41.327,157.885
C09848=1040.924,265.814,-110.225,171.447,41.328,157.885
C09849=1040.930,266.062,-110.255,171.451,41.330,157.886
C09850=1040.937,266.310,-110.285,171.453,41.332,157.886
C09851=1040.944,266.558,-110.315,171.456,41.334,157.887
C09852=1040.950,266.806,-110.346,171.459,41.335,157.887
C09853=1040.957,267.054,-110.376,171.462,41.338,157.888
C09854=1040.964,267.303,-110.406,171.466,41.339,157.889
C09855=1040.970,267.550,-110.436,171.468,41.341,157.889
C09856=1040.977,267.799,-110.466,171.472,41.343,157.890
C09857=1040.984,268.047,-110.497,171.475,41.345,157.890
C09858=1040.990,268.295,-110.527,171.478,41.346,157.891
C09859=1040.997,268.543,-110.558,171.481,41.349,157.892
C09860=1041.004,268.791,-110.588,171.485,41.350,157.892
C09861=1041.010,269.039,-110.617,171.487,41.352,157.893
C09862=1041.017,269.287,-110.649,171.491,41.354,157.893
C09863=1041.024,269.535,-110.679,171.494,41.356,157.894
C09864=1041.030,269.783,-110.709,171.497,41.358,157.894
C09865=1041.037,270.031,-110.739,171.500,41.359,157.895
C09866=1041.044,270.280,-110.770,171.504,41.361,157.896
C09867=1041.051,270.527,-110.801,171.506,41.363,157.896
C09868=1041.057,270.775,-110.831,171.510,41.365,157.897
C09869=1041.064,271.023,-110.862,171.512,41.367,157.897
C09870=1041.070,271.272,-110.892,171.516,41.369,157.898
C09871=1041.077,271.520,-110.924,171.519,41.371,157.898
C09872=1041.084,271.767,-110.953,171.522,41.372,157.899
C09873=1041.090,272.016,-110.984,171.525,41.374,157.900
C09874=1041.098,272.263,-111.015,171.529,41.377,157.900
C09875=1041.104,272.512,-111.046,171.531,41.378,157.901
C09876=1041.110,272.760,-111.076,171.535,41.380,157.901
C09877=1041.117,273.007,-111.107,171.538,41.382,157.902
C09878=1041.124,273.256,-111.138,171.541,41.384,157.903
C09879=1041.130,273.504,-111.169,171.545,41.386,157.903
C09880=1041.137,273.751,-111.199,171.548,41.387,157.904
C09881=1041.143,274.000,-111.229,171.551,41.389,157.904
C09882=1041.150,274.247,-111.261,171.554,41.392,157.905
C09883=1041.157,274.496,-111.291,171.558,41.393,157.906
C09884=1041.164,274.744,-111.322,171.560,41.395,157.906
C09885=1041.170,274.991,-111.353,171.564,41.397,157.907
C09886=1041.177,275.239,-111.384,171.567,41.399,157.907
C09887=1041.184,275.488,-111.414,171.570,41.401,157.908
C09888=1041.190,275.735,-111.446,171.574,41.403,157.909
C09889=1041.197,275.983,-111.477,171.577,41.405,157.909
C09890=1041.204,276.232,-111.507,171.580,41.406,157.910
C09891=1041.210,276.479,-111.538,171.583,41.409,157.910
C09892=1041.219,276.785,-111.577,171.587,41.411,157.911
C09893=1041.227,277.092,-111.615,171.592,41.413,157.912
C09894=1041.235,277.398,-111.653,171.596,41.416,157.913
C09895=1041.244,277.704,-111.691,171.600,41.418,157.913
C09896=1041.251,277.952,-111.723,171.603,41.420,157.914
C09897=1041.256,278.199,-111.753,171.606,41.422,157.915
C09898=1041.264,278.447,-111.784,171.610,41.424,157.915
C09899=1041.271,278.695,-111.815,171.613,41.426,157.916
C09900=1041.277,278.943,-111.847,171.616,41.428,157.916
C09901=1041.284,279.191,-111.878,171.620,41.430,157.917
C09902=1041.291,279.439,-111.909,171.622,41.432,157.918
C09903=1041.297,279.687,-111.940,171.626,41.434,157.918
C09904=1041.304,279.935,-111.972,171.630,41.436,157.919
C09905=1041.311,280.183,-112.003,171.633,41.438,157.920
C09906=1041.317,280.431,-112.035,171.636,41.440,157.920
C09907=1041.324,280.679,-112.065,171.640,41.442,157.921
C09908=1041.330,280.927,-112.096,171.643,41.444,157.921
C09909=1041.337,281.175,-112.128,171.646,41.446,157.922
C09910=1041.343,281.422,-112.159,171.649,41.448,157.923
C09911=1041.350,281.670,-112.191,171.653,41.450,157.923
C09912=1041.357,281.918,-112.222,171.657,41.452,157.924
C09913=1041.364,282.166,-112.254,171.659,41.454,157.925
C09914=1041.370,282.414,-112.285,171.663,41.456,157.925
C09915=1041.377,282.662,-112.317,171.667,41.458,157.926
C09916=1041.384,282.910,-112.348,171.669,41.460,157.927
C09917=1041.391,283.158,-112.379,171.673,41.462,157.927
C09918=1041.397,283.406,-112.411,171.677,41.464,157.928
C09919=1041.404,283.654,-112.442,171.680,41.466,157.928
C09920=1041.411,283.901,-112.474,171.683,41.468,157.929
C09921=1041.417,284.149,-112.505,171.687,41.470,157.930
C09922=1041.424,284.397,-112.537,171.690,41.472,157.930
C09923=1041.431,284.645,-112.568,171.694,41.474,157.931
C09924=1041.438,284.893,-112.599,171.697,41.476,157.932
C09925=1041.444,285.141,-112.631,171.701,41.478,157.932
C09926=1041.452,285.390,-112.663,171.704,41.480,157.933
C09927=1041.459,285.637,-112.695,171.707,41.482,157.934
C09928=1041.465,285.885,-112.726,171.711,41.484,157.934
C09929=1041.472,286.133,-112.758,171.715,41.486,157.935
C09930=1041.479,286.381,-112.789,171.718,41.488,157.936
C09931=1041.486,286.628,-112.821,171.721,41.490,157.936
C09932=1041.492,286.876,-112.852,171.725,41.492,157.937
C09933=1041.499,287.124,-112.884,171.728,41.494,157.937
C09934=1041.505,287.372,-112.916,171.732,41.496,157.938
C09935=1041.512,287.620,-112.948,171.735,41.498,157.939
C09936=1041.519,287.868,-112.979,171.739,41.500,157.939
C09937=1041.526,288.116,-113.011,171.742,41.503,157.940
C09938=1041.532,288.364,-113.044,171.746,41.505,157.941
C09939=1041.539,288.612,-113.075,171.749,41.507,157.941
C09940=1041.546,288.859,-113.107,171.753,41.509,157.942
C09941=1041.553,289.107,-113.139,171.756,41.511,157.943
C09942=1041.560,289.354,-113.171,171.760,41.513,157.944
C09943=1041.566,289.602,-113.203,171.763,41.515,157.944
C09944=1041.573,289.851,-113.235,171.767,41.517,157.945
C09945=1041.580,290.098,-113.267,171.770,41.520,157.945
C09946=1041.586,290.347,-113.299,171.774,41.522,157.946
C09947=1041.593,290.594,-113.331,171.777,41.524,157.947
C09948=1041.603,290.912,-113.372,171.783,41.527,157.948
C09949=1041.610,291.230,-113.413,171.786,41.529,157.949
C09950=1041.620,291.548,-113.454,171.791,41.532,157.949
C09951=1041.627,291.866,-113.495,171.795,41.534,157.950
C09952=1041.635,292.113,-113.527,171.799,41.537,157.951
C09953=1041.642,292.361,-113.560,171.803,41.539,157.952
C09954=1041.648,292.609,-113.592,171.807,41.541,157.952
C09955=1041.655,292.856,-113.624,171.810,41.543,157.953
C09956=1041.662,293.104,-113.655,171.813,41.545,157.954
C09957=1041.669,293.353,-113.689,171.817,41.547,157.954
C09958=1041.676,293.600,-113.721,171.821,41.550,157.955
C09959=1041.683,293.848,-113.752,171.825,41.552,157.956
C09960=1041.689,294.095,-113.785,171.828,41.554,157.957
C09961=1041.696,294.343,-113.817,171.832,41.556,157.957
C09962=1041.703,294.591,-113.850,171.835,41.559,157.958
C09963=1041.709,294.839,-113.882,171.839,41.561,157.959
C09964=1041.716,295.087,-113.914,171.843,41.563,157.959
C09965=1041.723,295.334,-113.947,171.846,41.565,157.960
C09966=1041.730,295.582,-113.980,171.850,41.567,157.961
C09967=1041.737,295.829,-114.012,171.854,41.569,157.961
C09968=1041.743,296.077,-114.044,171.857,41.572,157.962
C09969=1041.750,296.325,-114.078,171.861,41.574,157.963
C09970=1041.756,296.573,-114.110,171.864,41.576,157.964
C09971=1041.763,296.821,-114.142,171.868,41.579,157.964
C09972=1041.769,297.068,-114.174,171.872,41.581,157.965
C09973=1041.776,297.317,-114.208,171.876,41.583,157.966
C09974=1041.782,297.564,-114.240,171.879,41.585,157.966
C09975=1041.789,297.812,-114.273,171.883,41.588,157.967
C09976=1041.796,298.060,-114.306,171.886,41.590,157.968
C09977=1041.803,298.307,-114.338,171.890,41.592,157.969
C09978=1041.809,298.554,-114.372,171.894,41.595,157.969
C09979=1041.816,298.803,-114.405,171.898,41.597,157.970
C09980=1041.823,299.050,-114.437,171.902,41.599,157.971
C09981=1041.829,299.298,-114.470,171.906,41.601,157.972
C09982=1041.836,299.546,-114.503,171.909,41.604,157.972
C09983=1041.843,299.793,-114.536,171.912,41.606,157.973
C09984=1041.849,300.041,-114.568,171.916,41.609,157.974
C09985=1041.857,300.289,-114.601,171.920,41.611,157.975
C09986=1041.863,300.536,-114.634,171.924,41.613,157.975
C09987=1041.870,300.784,-114.667,171.928,41.615,157.976
C09988=1041.876,301.032,-114.700,171.932,41.618,157.977
C09989=1041.883,301.279,-114.733,171.935,41.620,157.977
C09990=1041.890,301.527,-114.765,171.939,41.622,157.978
C09991=1041.897,301.774,-114.799,171.943,41.624,157.979
C09992=1041.904,302.023,-114.832,171.947,41.627,157.980
C09993=1041.910,302.270,-114.865,171.951,41.629,157.980
C09994=1041.917,302.518,-114.899,171.955,41.632,157.981
C09995=1041.924,302.765,-114.931,171.958,41.634,157.982
C09996=1041.931,303.014,-114.964,171.961,41.636,157.983
//INST
///DATE 2021/06/17 10:57
///ATTR SC,RW,RJ
////FRAME ROBOT
///GROUP1 RB1
NOP
MOVL C00000 V=800.0 PL=0
MOVL C00001 V=800.0 PL=0
MOVL C00002 V=800.0 PL=0
MOVL C00003 V=800.0 PL=0
MOVL C00004 V=800.0 PL=0
MOVL C00005 V=800.0 PL=0
MOVL C00006 V=800.0 PL=0
MOVL C00007 V=800.0 PL=0
MOVL C00008 V=800.0 PL=0
MOVL C00009 V=800.0 PL=0
MOVL C00010 V=800.0 PL=0
MOVL C00011 V=800.0 PL=0
MOVL C00012 V=800.0 PL=0
MOVL C00013 V=800.0 PL=0
MOVL C00014 V=800.0 PL=0
MOVL C00015 V=800.0 PL=0
MOVL C00016 V=800.0 PL=0
MOVL C00017 V=800.0 PL=0
MOVL C00018 V=800.0 PL=0
MOVL C00019 V=800.0 PL=0
MOVL C00020 V=800.0 PL=0
MOVL C00021 V=800.0 PL=0
MOVL C00022 V=800.0 PL=0
MOVL C00023 V=800.0 PL=0
MOVL C00024 V=800.0 PL=0
MOVL C00025 V=800.0 PL=0
MOVL C00026 V=800.0 PL=0
MOVL C00027 V=800.0 PL=0
MOVL C00028 V=800.0 PL=0
MOVL C00029 V=800.0 PL=0
MOVL C00030 V=800.0 PL=0
MOVL C00031 V=800.0 PL=0
MOVL C00032 V=800.0 PL=0
MOVL C00033 V=800.0 PL=0
MOVL C00034 V=800.0 PL=0
MOVL C00035 V=800.0 PL=0
MOVL C00036 V=800.0 PL=0
MOVL C00037 V=800.0 PL=0
MOVL C00038 V=800.0 PL=0
MOVL C00039 V=800.0 PL=0
MOVL C00040 V=800.0 PL=0
MOVL C00041 V=800.0 PL=0
MOVL C00042 V=800.0 PL=0
MOVL C00043 V=800.0 PL=0
MOVL C00044 V=800.0 PL=0
MOVL C00045 V=800.0 PL=0
MOVL C00046 V=800.0 PL=0
MOVL C00047 V=800.0 PL=0
MOVL C00048 V=800.0 PL=0
MOVL C00049 V=800.0 PL=0
MOVL C00050 V=800.0 PL=0
MOVL C00051 V=800.0 PL=0
MOVL C00052 V=800.0 PL=0
MOVL C00053 V=800.0 PL=0
MOVL C00054 V=800.0 PL=0
MOVL C00055 V=800.0 PL=0
MOVL C00056 V=800.0 PL=0
MOVL C00057 V=800.0 PL=0
MOVL C00058 V=800.0 PL=0
MOVL C00059 V=800.0 PL=0
MOVL C00060 V=800.0 PL=0
MOVL C00061 V=800.0 PL=0
MOVL C00062 V=800.0 PL=0
MOVL C00063 V=800.0 PL=0
MOVL C00064 V=800.0 PL=0
MOVL C00065 V=800.0 PL=0
MOVL C00066 V=800.0 PL=0
MOVL C00067 V=800.0 PL=0
MOVL C00068 V=800.0 PL=0
MOVL C00069 V=800.0 PL=0
MOVL C00070 V=800.0 PL=0
MOVL C00071 V=800.0 PL=0
MOVL C00072 V=800.0 PL=0
MOVL C00073 V=800.0 PL=0
MOVL C00074 V=800.0 PL=0
MOVL C00075 V=800.0 PL=0
MOVL C00076 V=800.0 PL=0
MOVL C00077 V=800.0 PL=0
MOVL C00078 V=800.0 PL=0
MOVL C00079 V=800.0 PL=0
MOVL C00080 V=800.0 PL=0
MOVL C00081 V=800.0 PL=0
MOVL C00082 V=800.0 PL=0
MOVL C00083 V=800.0 PL=0
MOVL C00084 V=800.0 PL=0
MOVL C00085 V=800.0 PL=0
MOVL C00086 V=800.0 PL=0
MOVL C00087 V=800.0 PL=0
MOVL C00088 V=800.0 PL=0
MOVL C00089 V=800.0 PL=0
MOVL C00090 V=800.0 PL=0
MOVL C00091 V=800.0 PL=0
MOVL C00092 V=800.0 PL=0
MOVL C00093 V=800.0 PL=0
MOVL C00094 V=800.0 PL=0
MOVL C00095 V=800.0 PL=0
MOVL C00096 V=800.0 PL=0
MOVL C00097 V=800.0 PL=0
MOVL C00098 V=800.0 PL=0
MOVL C00099 V=800.0 PL=0
MOVL C00100 V=800.0 PL=0
MOVL C00101 V=800.0 PL=0
MOVL C00102 V=800.0 PL=0
MOVL C00103 V=800.0 PL=0
MOVL C00104 V=800.0 PL=0
MOVL C00105 V=800.0 PL=0
MOVL C00106 V=800.0 PL=0
MOVL C00107 V=800.0 PL=0
MOVL C00108 V=800.0 PL=0
MOVL C00109 V=800.0 PL=0
MOVL C00110 V=800.0 PL=0
MOVL C00111 V=800.0 PL=0
MOVL C00112 V=800.0 PL=0
MOVL C00113 V=800.0 PL=0
MOVL C00114 V=800.0 PL=0
MOVL C00115 V=800.0 PL=0
MOVL C00116 V=800.0 PL=0
MOVL C00117 V=800.0 PL=0
MOVL C00118 V=800.0 PL=0
MOVL C00119 V=800.0 PL=0
MOVL C00120 V=800.0 PL=0
MOVL C00121 V=800.0 PL=0
MOVL C00122 V=800.0 PL=0
MOVL C00123 V=800.0 PL=0
MOVL C00124 V=800.0 PL=0
MOVL C00125 V=800.0 PL=0
MOVL C00126 V=800.0 PL=0
MOVL C00127 V=800.0 PL=0
MOVL C00128 V=800.0 PL=0
MOVL C00129 V=800.0 PL=0
MOVL C00130 V=800.0 PL=0
MOVL C00131 V=800.0 PL=0
MOVL C00132 V=800.0 PL=0
MOVL C00133 V=800.0 PL=0
MOVL C00134 V=800.0 PL=0
MOVL C00135 V=800.0 PL=0
MOVL C00136 V=800.0 PL=0
MOVL C00137 V=800.0 PL=0
MOVL C00138 V=800.0 PL=0
MOVL C00139 V=800.0 PL=0
MOVL C00140 V=800.0 PL=0
MOVL C00141 V=800.0 PL=0
MOVL C00142 V=800.0 PL=0
MOVL C00143 V=800.0 PL=0
MOVL C00144 V=800.0 PL=0
MOVL C00145 V=800.0 PL=0
MOVL C00146 V=800.0 PL=0
MOVL C00147 V=800.0 PL=0
MOVL C00148 V=800.0 PL=0
MOVL C00149 V=800.0 PL=0
MOVL C00150 V=800.0 PL=0
MOVL C00151 V=800.0 PL=0
MOVL C00152 V=800.0 PL=0
MOVL C00153 V=800.0 PL=0
MOVL C00154 V=800.0 PL=0
MOVL C00155 V=800.0 PL=0
MOVL C00156 V=800.0 PL=0
MOVL C00157 V=800.0 PL=0
MOVL C00158 V=800.0 PL=0
MOVL C00159 V=800.0 PL=0
MOVL C00160 V=800.0 PL=0
MOVL C00161 V=800.0 PL=0
MOVL C00162 V=800.0 PL=0
MOVL C00163 V=800.0 PL=0
MOVL C00164 V=800.0 PL=0
MOVL C00165 V=800.0 PL=0
MOVL C00166 V=800.0 PL=0
MOVL C00167 V=800.0 PL=0
MOVL C00168 V=800.0 PL=0
MOVL C00169 V=800.0 PL=0
MOVL C00170 V=800.0 PL=0
MOVL C00171 V=800.0 PL=0
MOVL C00172 V=800.0 PL=0
MOVL C00173 V=800.0 PL=0
MOVL C00174 V=800.0 PL=0
MOVL C00175 V=800.0 PL=0
MOVL C00176 V=800.0 PL=0
MOVL C00177 V=800.0 PL=0
MOVL C00178 V=800.0 PL=0
MOVL C00179 V=800.0 PL=0
MOVL C00180 V=800.0 PL=0
MOVL C00181 V=800.0 PL=0
MOVL C00182 V=800.0 PL=0
MOVL C00183 V=800.0 PL=0
MOVL C00184 V=800.0 PL=0
MOVL C00185 V=800.0 PL=0
MOVL C00186 V=800.0 PL=0
MOVL C00187 V=800.0 PL=0
MOVL C00188 V=800.0 PL=0
MOVL C00189 V=800.0 PL=0
MOVL C00190 V=800.0 PL=0
MOVL C00191 V=800.0 PL=0
MOVL C00192 V=800.0 PL=0
MOVL C00193 V=800.0 PL=0
MOVL C00194 V=800.0 PL=0
MOVL C00195 V=800.0 PL=0
MOVL C00196 V=800.0 PL=0
MOVL C00197 V=800.0 PL=0
MOVL C00198 V=800.0 PL=0
MOVL C00199 V=800.0 PL=0
MOVL C00200 V=800.0 PL=0
MOVL C00201 V=800.0 PL=0
MOVL C00202 V=800.0 PL=0
MOVL C00203 V=800.0 PL=0
MOVL C00204 V=800.0 PL=0
MOVL C00205 V=800.0 PL=0
MOVL C00206 V=800.0 PL=0
MOVL C00207 V=800.0 PL=0
MOVL C00208 V=800.0 PL=0
MOVL C00209 V=800.0 PL=0
MOVL C00210 V=800.0 PL=0
MOVL C00211 V=800.0 PL=0
MOVL C00212 V=800.0 PL=0
MOVL C00213 V=800.0 PL=0
MOVL C00214 V=800.0 PL=0
MOVL C00215 V=800.0 PL=0
MOVL C00216 V=800.0 PL=0
MOVL C00217 V=800.0 PL=0
MOVL C00218 V=800.0 PL=0
MOVL C00219 V=800.0 PL=0
MOVL C00220 V=800.0 PL=0
MOVL C00221 V=800.0 PL=0
MOVL C00222 V=800.0 PL=0
MOVL C00223 V=800.0 PL=0
MOVL C00224 V=800.0 PL=0
MOVL C00225 V=800.0 PL=0
MOVL C00226 V=800.0 PL=0
MOVL C00227 V=800.0 PL=0
MOVL C00228 V=800.0 PL=0
MOVL C00229 V=800.0 PL=0
MOVL C00230 V=800.0 PL=0
MOVL C00231 V=800.0 PL=0
MOVL C00232 V=800.0 PL=0
MOVL C00233 V=800.0 PL=0
MOVL C00234 V=800.0 PL=0
MOVL C00235 V=800.0 PL=0
MOVL C00236 V=800.0 PL=0
MOVL C00237 V=800.0 PL=0
MOVL C00238 V=800.0 PL=0
MOVL C00239 V=800.0 PL=0
MOVL C00240 V=800.0 PL=0
MOVL C00241 V=800.0 PL=0
MOVL C00242 V=800.0 PL=0
MOVL C00243 V=800.0 PL=0
MOVL C00244 V=800.0 PL=0
MOVL C00245 V=800.0 PL=0
MOVL C00246 V=800.0 PL=0
MOVL C00247 V=800.0 PL=0
MOVL C00248 V=800.0 PL=0
MOVL C00249 V=800.0 PL=0
MOVL C00250 V=800.0 PL=0
MOVL C00251 V=800.0 PL=0
MOVL C00252 V=800.0 PL=0
MOVL C00253 V=800.0 PL=0
MOVL C00254 V=800.0 PL=0
MOVL C00255 V=800.0 PL=0
MOVL C00256 V=800.0 PL=0
MOVL C00257 V=800.0 PL=0
MOVL C00258 V=800.0 PL=0
MOVL C00259 V=800.0 PL=0
MOVL C00260 V=800.0 PL=0
MOVL C00261 V=800.0 PL=0
MOVL C00262 V=800.0 PL=0
MOVL C00263 V=800.0 PL=0
MOVL C00264 V=800.0 PL=0
MOVL C00265 V=800.0 PL=0
MOVL C00266 V=800.0 PL=0
MOVL C00267 V=800.0 PL=0
MOVL C00268 V=800.0 PL=0
MOVL C00269 V=800.0 PL=0
MOVL C00270 V=800.0 PL=0
MOVL C00271 V=800.0 PL=0
MOVL C00272 V=800.0 PL=0
MOVL C00273 V=800.0 PL=0
MOVL C00274 V=800.0 PL=0
MOVL C00275 V=800.0 PL=0
MOVL C00276 V=800.0 PL=0
MOVL C00277 V=800.0 PL=0
MOVL C00278 V=800.0 PL=0
MOVL C00279 V=800.0 PL=0
MOVL C00280 V=800.0 PL=0
MOVL C00281 V=800.0 PL=0
MOVL C00282 V=800.0 PL=0
MOVL C00283 V=800.0 PL=0
MOVL C00284 V=800.0 PL=0
MOVL C00285 V=800.0 PL=0
MOVL C00286 V=800.0 PL=0
MOVL C00287 V=800.0 PL=0
MOVL C00288 V=800.0 PL=0
MOVL C00289 V=800.0 PL=0
MOVL C00290 V=800.0 PL=0
MOVL C00291 V=800.0 PL=0
MOVL C00292 V=800.0 PL=0
MOVL C00293 V=800.0 PL=0
MOVL C00294 V=800.0 PL=0
MOVL C00295 V=800.0 PL=0
MOVL C00296 V=800.0 PL=0
MOVL C00297 V=800.0 PL=0
MOVL C00298 V=800.0 PL=0
MOVL C00299 V=800.0 PL=0
MOVL C00300 V=800.0 PL=0
MOVL C00301 V=800.0 PL=0
MOVL C00302 V=800.0 PL=0
MOVL C00303 V=800.0 PL=0
MOVL C00304 V=800.0 PL=0
MOVL C00305 V=800.0 PL=0
MOVL C00306 V=800.0 PL=0
MOVL C00307 V=800.0 PL=0
MOVL C00308 V=800.0 PL=0
MOVL C00309 V=800.0 PL=0
MOVL C00310 V=800.0 PL=0
MOVL C00311 V=800.0 PL=0
MOVL C00312 V=800.0 PL=0
MOVL C00313 V=800.0 PL=0
MOVL C00314 V=800.0 PL=0
MOVL C00315 V=800.0 PL=0
MOVL C00316 V=800.0 PL=0
MOVL C00317 V=800.0 PL=0
MOVL C00318 V=800.0 PL=0
MOVL C00319 V=800.0 PL=0
MOVL C00320 V=800.0 PL=0
MOVL C00321 V=800.0 PL=0
MOVL C00322 V=800.0 PL=0
MOVL C00323 V=800.0 PL=0
MOVL C00324 V=800.0 PL=0
MOVL C00325 V=800.0 PL=0
MOVL C00326 V=800.0 PL=0
MOVL C00327 V=800.0 PL=0
MOVL C00328 V=800.0 PL=0
MOVL C00329 V=800.0 PL=0
MOVL C00330 V=800.0 PL=0
MOVL C00331 V=800.0 PL=0
MOVL C00332 V=800.0 PL=0
MOVL C00333 V=800.0 PL=0
MOVL C00334 V=800.0 PL=0
MOVL C00335 V=800.0 PL=0
MOVL C00336 V=800.0 PL=0
MOVL C00337 V=800.0 PL=0
MOVL C00338 V=800.0 PL=0
MOVL C00339 V=800.0 PL=0
MOVL C00340 V=800.0 PL=0
MOVL C00341 V=800.0 PL=0
MOVL C00342 V=800.0 PL=0
MOVL C00343 V=800.0 PL=0
MOVL C00344 V=800.0 PL=0
MOVL C00345 V=800.0 PL=0
MOVL C00346 V=800.0 PL=0
MOVL C00347 V=800.0 PL=0
MOVL C00348 V=800.0 PL=0
MOVL C00349 V=800.0 PL=0
MOVL C00350 V=800.0 PL=0
MOVL C00351 V=800.0 PL=0
MOVL C00352 V=800.0 PL=0
MOVL C00353 V=800.0 PL=0
MOVL C00354 V=800.0 PL=0
MOVL C00355 V=800.0 PL=0
MOVL C00356 V=800.0 PL=0
MOVL C00357 V=800.0 PL=0
MOVL C00358 V=800.0 PL=0
MOVL C00359 V=800.0 PL=0
MOVL C00360 V=800.0 PL=0
MOVL C00361 V=800.0 PL=0
MOVL C00362 V=800.0 PL=0
MOVL C00363 V=800.0 PL=0
MOVL C00364 V=800.0 PL=0
MOVL C00365 V=800.0 PL=0
MOVL C00366 V=800.0 PL=0
MOVL C00367 V=800.0 PL=0
MOVL C00368 V=800.0 PL=0
MOVL C00369 V=800.0 PL=0
MOVL C00370 V=800.0 PL=0
MOVL C00371 V=800.0 PL=0
MOVL C00372 V=800.0 PL=0
MOVL C00373 V=800.0 PL=0
MOVL C00374 V=800.0 PL=0
MOVL C00375 V=800.0 PL=0
MOVL C00376 V=800.0 PL=0
MOVL C00377 V=800.0 PL=0
MOVL C00378 V=800.0 PL=0
MOVL C00379 V=800.0 PL=0
MOVL C00380 V=800.0 PL=0
MOVL C00381 V=800.0 PL=0
MOVL C00382 V=800.0 PL=0
MOVL C00383 V=800.0 PL=0
MOVL C00384 V=800.0 PL=0
MOVL C00385 V=800.0 PL=0
MOVL C00386 V=800.0 PL=0
MOVL C00387 V=800.0 PL=0
MOVL C00388 V=800.0 PL=0
MOVL C00389 V=800.0 PL=0
MOVL C00390 V=800.0 PL=0
MOVL C00391 V=800.0 PL=0
MOVL C00392 V=800.0 PL=0
MOVL C00393 V=800.0 PL=0
MOVL C00394 V=800.0 PL=0
MOVL C00395 V=800.0 PL=0
MOVL C00396 V=800.0 PL=0
MOVL C00397 V=800.0 PL=0
MOVL C00398 V=800.0 PL=0
MOVL C00399 V=800.0 PL=0
MOVL C00400 V=800.0 PL=0
MOVL C00401 V=800.0 PL=0
MOVL C00402 V=800.0 PL=0
MOVL C00403 V=800.0 PL=0
MOVL C00404 V=800.0 PL=0
MOVL C00405 V=800.0 PL=0
MOVL C00406 V=800.0 PL=0
MOVL C00407 V=800.0 PL=0
MOVL C00408 V=800.0 PL=0
MOVL C00409 V=800.0 PL=0
MOVL C00410 V=800.0 PL=0
MOVL C00411 V=800.0 PL=0
MOVL C00412 V=800.0 PL=0
MOVL C00413 V=800.0 PL=0
MOVL C00414 V=800.0 PL=0
MOVL C00415 V=800.0 PL=0
MOVL C00416 V=800.0 PL=0
MOVL C00417 V=800.0 PL=0
MOVL C00418 V=800.0 PL=0
MOVL C00419 V=800.0 PL=0
MOVL C00420 V=800.0 PL=0
MOVL C00421 V=800.0 PL=0
MOVL C00422 V=800.0 PL=0
MOVL C00423 V=800.0 PL=0
MOVL C00424 V=800.0 PL=0
MOVL C00425 V=800.0 PL=0
MOVL C00426 V=800.0 PL=0
MOVL C00427 V=800.0 PL=0
MOVL C00428 V=800.0 PL=0
MOVL C00429 V=800.0 PL=0
MOVL C00430 V=800.0 PL=0
MOVL C00431 V=800.0 PL=0
MOVL C00432 V=800.0 PL=0
MOVL C00433 V=800.0 PL=0
MOVL C00434 V=800.0 PL=0
MOVL C00435 V=800.0 PL=0
MOVL C00436 V=800.0 PL=0
MOVL C00437 V=800.0 PL=0
MOVL C00438 V=800.0 PL=0
MOVL C00439 V=800.0 PL=0
MOVL C00440 V=800.0 PL=0
MOVL C00441 V=800.0 PL=0
MOVL C00442 V=800.0 PL=0
MOVL C00443 V=800.0 PL=0
MOVL C00444 V=800.0 PL=0
MOVL C00445 V=800.0 PL=0
MOVL C00446 V=800.0 PL=0
MOVL C00447 V=800.0 PL=0
MOVL C00448 V=800.0 PL=0
MOVL C00449 V=800.0 PL=0
MOVL C00450 V=800.0 PL=0
MOVL C00451 V=800.0 PL=0
MOVL C00452 V=800.0 PL=0
MOVL C00453 V=800.0 PL=0
MOVL C00454 V=800.0 PL=0
MOVL C00455 V=800.0 PL=0
MOVL C00456 V=800.0 PL=0
MOVL C00457 V=800.0 PL=0
MOVL C00458 V=800.0 PL=0
MOVL C00459 V=800.0 PL=0
MOVL C00460 V=800.0 PL=0
MOVL C00461 V=800.0 PL=0
MOVL C00462 V=800.0 PL=0
MOVL C00463 V=800.0 PL=0
MOVL C00464 V=800.0 PL=0
MOVL C00465 V=800.0 PL=0
MOVL C00466 V=800.0 PL=0
MOVL C00467 V=800.0 PL=0
MOVL C00468 V=800.0 PL=0
MOVL C00469 V=800.0 PL=0
MOVL C00470 V=800.0 PL=0
MOVL C00471 V=800.0 PL=0
MOVL C00472 V=800.0 PL=0
MOVL C00473 V=800.0 PL=0
MOVL C00474 V=800.0 PL=0
MOVL C00475 V=800.0 PL=0
MOVL C00476 V=800.0 PL=0
MOVL C00477 V=800.0 PL=0
MOVL C00478 V=800.0 PL=0
MOVL C00479 V=800.0 PL=0
MOVL C00480 V=800.0 PL=0
MOVL C00481 V=800.0 PL=0
MOVL C00482 V=800.0 PL=0
MOVL C00483 V=800.0 PL=0
MOVL C00484 V=800.0 PL=0
MOVL C00485 V=800.0 PL=0
MOVL C00486 V=800.0 PL=0
MOVL C00487 V=800.0 PL=0
MOVL C00488 V=800.0 PL=0
MOVL C00489 V=800.0 PL=0
MOVL C00490 V=800.0 PL=0
MOVL C00491 V=800.0 PL=0
MOVL C00492 V=800.0 PL=0
MOVL C00493 V=800.0 PL=0
MOVL C00494 V=800.0 PL=0
MOVL C00495 V=800.0 PL=0
MOVL C00496 V=800.0 PL=0
MOVL C00497 V=800.0 PL=0
MOVL C00498 V=800.0 PL=0
MOVL C00499 V=800.0 PL=0
MOVL C00500 V=800.0 PL=0
MOVL C00501 V=800.0 PL=0
MOVL C00502 V=800.0 PL=0
MOVL C00503 V=800.0 PL=0
MOVL C00504 V=800.0 PL=0
MOVL C00505 V=800.0 PL=0
MOVL C00506 V=800.0 PL=0
MOVL C00507 V=800.0 PL=0
MOVL C00508 V=800.0 PL=0
MOVL C00509 V=800.0 PL=0
MOVL C00510 V=800.0 PL=0
MOVL C00511 V=800.0 PL=0
MOVL C00512 V=800.0 PL=0
MOVL C00513 V=800.0 PL=0
MOVL C00514 V=800.0 PL=0
MOVL C00515 V=800.0 PL=0
MOVL C00516 V=800.0 PL=0
MOVL C00517 V=800.0 PL=0
MOVL C00518 V=800.0 PL=0
MOVL C00519 V=800.0 PL=0
MOVL C00520 V=800.0 PL=0
MOVL C00521 V=800.0 PL=0
MOVL C00522 V=800.0 PL=0
MOVL C00523 V=800.0 PL=0
MOVL C00524 V=800.0 PL=0
MOVL C00525 V=800.0 PL=0
MOVL C00526 V=800.0 PL=0
MOVL C00527 V=800.0 PL=0
MOVL C00528 V=800.0 PL=0
MOVL C00529 V=800.0 PL=0
MOVL C00530 V=800.0 PL=0
MOVL C00531 V=800.0 PL=0
MOVL C00532 V=800.0 PL=0
MOVL C00533 V=800.0 PL=0
MOVL C00534 V=800.0 PL=0
MOVL C00535 V=800.0 PL=0
MOVL C00536 V=800.0 PL=0
MOVL C00537 V=800.0 PL=0
MOVL C00538 V=800.0 PL=0
MOVL C00539 V=800.0 PL=0
MOVL C00540 V=800.0 PL=0
MOVL C00541 V=800.0 PL=0
MOVL C00542 V=800.0 PL=0
MOVL C00543 V=800.0 PL=0
MOVL C00544 V=800.0 PL=0
MOVL C00545 V=800.0 PL=0
MOVL C00546 V=800.0 PL=0
MOVL C00547 V=800.0 PL=0
MOVL C00548 V=800.0 PL=0
MOVL C00549 V=800.0 PL=0
MOVL C00550 V=800.0 PL=0
MOVL C00551 V=800.0 PL=0
MOVL C00552 V=800.0 PL=0
MOVL C00553 V=800.0 PL=0
MOVL C00554 V=800.0 PL=0
MOVL C00555 V=800.0 PL=0
MOVL C00556 V=800.0 PL=0
MOVL C00557 V=800.0 PL=0
MOVL C00558 V=800.0 PL=0
MOVL C00559 V=800.0 PL=0
MOVL C00560 V=800.0 PL=0
MOVL C00561 V=800.0 PL=0
MOVL C00562 V=800.0 PL=0
MOVL C00563 V=800.0 PL=0
MOVL C00564 V=800.0 PL=0
MOVL C00565 V=800.0 PL=0
MOVL C00566 V=800.0 PL=0
MOVL C00567 V=800.0 PL=0
MOVL C00568 V=800.0 PL=0
MOVL C00569 V=800.0 PL=0
MOVL C00570 V=800.0 PL=0
MOVL C00571 V=800.0 PL=0
MOVL C00572 V=800.0 PL=0
MOVL C00573 V=800.0 PL=0
MOVL C00574 V=800.0 PL=0
MOVL C00575 V=800.0 PL=0
MOVL C00576 V=800.0 PL=0
MOVL C00577 V=800.0 PL=0
MOVL C00578 V=800.0 PL=0
MOVL C00579 V=800.0 PL=0
MOVL C00580 V=800.0 PL=0
MOVL C00581 V=800.0 PL=0
MOVL C00582 V=800.0 PL=0
MOVL C00583 V=800.0 PL=0
MOVL C00584 V=800.0 PL=0
MOVL C00585 V=800.0 PL=0
MOVL C00586 V=800.0 PL=0
MOVL C00587 V=800.0 PL=0
MOVL C00588 V=800.0 PL=0
MOVL C00589 V=800.0 PL=0
MOVL C00590 V=800.0 PL=0
MOVL C00591 V=800.0 PL=0
MOVL C00592 V=800.0 PL=0
MOVL C00593 V=800.0 PL=0
MOVL C00594 V=800.0 PL=0
MOVL C00595 V=800.0 PL=0
MOVL C00596 V=800.0 PL=0
MOVL C00597 V=800.0 PL=0
MOVL C00598 V=800.0 PL=0
MOVL C00599 V=800.0 PL=0
MOVL C00600 V=800.0 PL=0
MOVL C00601 V=800.0 PL=0
MOVL C00602 V=800.0 PL=0
MOVL C00603 V=800.0 PL=0
MOVL C00604 V=800.0 PL=0
MOVL C00605 V=800.0 PL=0
MOVL C00606 V=800.0 PL=0
MOVL C00607 V=800.0 PL=0
MOVL C00608 V=800.0 PL=0
MOVL C00609 V=800.0 PL=0
MOVL C00610 V=800.0 PL=0
MOVL C00611 V=800.0 PL=0
MOVL C00612 V=800.0 PL=0
MOVL C00613 V=800.0 PL=0
MOVL C00614 V=800.0 PL=0
MOVL C00615 V=800.0 PL=0
MOVL C00616 V=800.0 PL=0
MOVL C00617 V=800.0 PL=0
MOVL C00618 V=800.0 PL=0
MOVL C00619 V=800.0 PL=0
MOVL C00620 V=800.0 PL=0
MOVL C00621 V=800.0 PL=0
MOVL C00622 V=800.0 PL=0
MOVL C00623 V=800.0 PL=0
MOVL C00624 V=800.0 PL=0
MOVL C00625 V=800.0 PL=0
MOVL C00626 V=800.0 PL=0
MOVL C00627 V=800.0 PL=0
MOVL C00628 V=800.0 PL=0
MOVL C00629 V=800.0 PL=0
MOVL C00630 V=800.0 PL=0
MOVL C00631 V=800.0 PL=0
MOVL C00632 V=800.0 PL=0
MOVL C00633 V=800.0 PL=0
MOVL C00634 V=800.0 PL=0
MOVL C00635 V=800.0 PL=0
MOVL C00636 V=800.0 PL=0
MOVL C00637 V=800.0 PL=0
MOVL C00638 V=800.0 PL=0
MOVL C00639 V=800.0 PL=0
MOVL C00640 V=800.0 PL=0
MOVL C00641 V=800.0 PL=0
MOVL C00642 V=800.0 PL=0
MOVL C00643 V=800.0 PL=0
MOVL C00644 V=800.0 PL=0
MOVL C00645 V=800.0 PL=0
MOVL C00646 V=800.0 PL=0
MOVL C00647 V=800.0 PL=0
MOVL C00648 V=800.0 PL=0
MOVL C00649 V=800.0 PL=0
MOVL C00650 V=800.0 PL=0
MOVL C00651 V=800.0 PL=0
MOVL C00652 V=800.0 PL=0
MOVL C00653 V=800.0 PL=0
MOVL C00654 V=800.0 PL=0
MOVL C00655 V=800.0 PL=0
MOVL C00656 V=800.0 PL=0
MOVL C00657 V=800.0 PL=0
MOVL C00658 V=800.0 PL=0
MOVL C00659 V=800.0 PL=0
MOVL C00660 V=800.0 PL=0
MOVL C00661 V=800.0 PL=0
MOVL C00662 V=800.0 PL=0
MOVL C00663 V=800.0 PL=0
MOVL C00664 V=800.0 PL=0
MOVL C00665 V=800.0 PL=0
MOVL C00666 V=800.0 PL=0
MOVL C00667 V=800.0 PL=0
MOVL C00668 V=800.0 PL=0
MOVL C00669 V=800.0 PL=0
MOVL C00670 V=800.0 PL=0
MOVL C00671 V=800.0 PL=0
MOVL C00672 V=800.0 PL=0
MOVL C00673 V=800.0 PL=0
MOVL C00674 V=800.0 PL=0
MOVL C00675 V=800.0 PL=0
MOVL C00676 V=800.0 PL=0
MOVL C00677 V=800.0 PL=0
MOVL C00678 V=800.0 PL=0
MOVL C00679 V=800.0 PL=0
MOVL C00680 V=800.0 PL=0
MOVL C00681 V=800.0 PL=0
MOVL C00682 V=800.0 PL=0
MOVL C00683 V=800.0 PL=0
MOVL C00684 V=800.0 PL=0
MOVL C00685 V=800.0 PL=0
MOVL C00686 V=800.0 PL=0
MOVL C00687 V=800.0 PL=0
MOVL C00688 V=800.0 PL=0
MOVL C00689 V=800.0 PL=0
MOVL C00690 V=800.0 PL=0
MOVL C00691 V=800.0 PL=0
MOVL C00692 V=800.0 PL=0
MOVL C00693 V=800.0 PL=0
MOVL C00694 V=800.0 PL=0
MOVL C00695 V=800.0 PL=0
MOVL C00696 V=800.0 PL=0
MOVL C00697 V=800.0 PL=0
MOVL C00698 V=800.0 PL=0
MOVL C00699 V=800.0 PL=0
MOVL C00700 V=800.0 PL=0
MOVL C00701 V=800.0 PL=0
MOVL C00702 V=800.0 PL=0
MOVL C00703 V=800.0 PL=0
MOVL C00704 V=800.0 PL=0
MOVL C00705 V=800.0 PL=0
MOVL C00706 V=800.0 PL=0
MOVL C00707 V=800.0 PL=0
MOVL C00708 V=800.0 PL=0
MOVL C00709 V=800.0 PL=0
MOVL C00710 V=800.0 PL=0
MOVL C00711 V=800.0 PL=0
MOVL C00712 V=800.0 PL=0
MOVL C00713 V=800.0 PL=0
MOVL C00714 V=800.0 PL=0
MOVL C00715 V=800.0 PL=0
MOVL C00716 V=800.0 PL=0
MOVL C00717 V=800.0 PL=0
MOVL C00718 V=800.0 PL=0
MOVL C00719 V=800.0 PL=0
MOVL C00720 V=800.0 PL=0
MOVL C00721 V=800.0 PL=0
MOVL C00722 V=800.0 PL=0
MOVL C00723 V=800.0 PL=0
MOVL C00724 V=800.0 PL=0
MOVL C00725 V=800.0 PL=0
MOVL C00726 V=800.0 PL=0
MOVL C00727 V=800.0 PL=0
MOVL C00728 V=800.0 PL=0
MOVL C00729 V=800.0 PL=0
MOVL C00730 V=800.0 PL=0
MOVL C00731 V=800.0 PL=0
MOVL C00732 V=800.0 PL=0
MOVL C00733 V=800.0 PL=0
MOVL C00734 V=800.0 PL=0
MOVL C00735 V=800.0 PL=0
MOVL C00736 V=800.0 PL=0
MOVL C00737 V=800.0 PL=0
MOVL C00738 V=800.0 PL=0
MOVL C00739 V=800.0 PL=0
MOVL C00740 V=800.0 PL=0
MOVL C00741 V=800.0 PL=0
MOVL C00742 V=800.0 PL=0
MOVL C00743 V=800.0 PL=0
MOVL C00744 V=800.0 PL=0
MOVL C00745 V=800.0 PL=0
MOVL C00746 V=800.0 PL=0
MOVL C00747 V=800.0 PL=0
MOVL C00748 V=800.0 PL=0
MOVL C00749 V=800.0 PL=0
MOVL C00750 V=800.0 PL=0
MOVL C00751 V=800.0 PL=0
MOVL C00752 V=800.0 PL=0
MOVL C00753 V=800.0 PL=0
MOVL C00754 V=800.0 PL=0
MOVL C00755 V=800.0 PL=0
MOVL C00756 V=800.0 PL=0
MOVL C00757 V=800.0 PL=0
MOVL C00758 V=800.0 PL=0
MOVL C00759 V=800.0 PL=0
MOVL C00760 V=800.0 PL=0
MOVL C00761 V=800.0 PL=0
MOVL C00762 V=800.0 PL=0
MOVL C00763 V=800.0 PL=0
MOVL C00764 V=800.0 PL=0
MOVL C00765 V=800.0 PL=0
MOVL C00766 V=800.0 PL=0
MOVL C00767 V=800.0 PL=0
MOVL C00768 V=800.0 PL=0
MOVL C00769 V=800.0 PL=0
MOVL C00770 V=800.0 PL=0
MOVL C00771 V=800.0 PL=0
MOVL C00772 V=800.0 PL=0
MOVL C00773 V=800.0 PL=0
MOVL C00774 V=800.0 PL=0
MOVL C00775 V=800.0 PL=0
MOVL C00776 V=800.0 PL=0
MOVL C00777 V=800.0 PL=0
MOVL C00778 V=800.0 PL=0
MOVL C00779 V=800.0 PL=0
MOVL C00780 V=800.0 PL=0
MOVL C00781 V=800.0 PL=0
MOVL C00782 V=800.0 PL=0
MOVL C00783 V=800.0 PL=0
MOVL C00784 V=800.0 PL=0
MOVL C00785 V=800.0 PL=0
MOVL C00786 V=800.0 PL=0
MOVL C00787 V=800.0 PL=0
MOVL C00788 V=800.0 PL=0
MOVL C00789 V=800.0 PL=0
MOVL C00790 V=800.0 PL=0
MOVL C00791 V=800.0 PL=0
MOVL C00792 V=800.0 PL=0
MOVL C00793 V=800.0 PL=0
MOVL C00794 V=800.0 PL=0
MOVL C00795 V=800.0 PL=0
MOVL C00796 V=800.0 PL=0
MOVL C00797 V=800.0 PL=0
MOVL C00798 V=800.0 PL=0
MOVL C00799 V=800.0 PL=0
MOVL C00800 V=800.0 PL=0
MOVL C00801 V=800.0 PL=0
MOVL C00802 V=800.0 PL=0
MOVL C00803 V=800.0 PL=0
MOVL C00804 V=800.0 PL=0
MOVL C00805 V=800.0 PL=0
MOVL C00806 V=800.0 PL=0
MOVL C00807 V=800.0 PL=0
MOVL C00808 V=800.0 PL=0
MOVL C00809 V=800.0 PL=0
MOVL C00810 V=800.0 PL=0
MOVL C00811 V=800.0 PL=0
MOVL C00812 V=800.0 PL=0
MOVL C00813 V=800.0 PL=0
MOVL C00814 V=800.0 PL=0
MOVL C00815 V=800.0 PL=0
MOVL C00816 V=800.0 PL=0
MOVL C00817 V=800.0 PL=0
MOVL C00818 V=800.0 PL=0
MOVL C00819 V=800.0 PL=0
MOVL C00820 V=800.0 PL=0
MOVL C00821 V=800.0 PL=0
MOVL C00822 V=800.0 PL=0
MOVL C00823 V=800.0 PL=0
MOVL C00824 V=800.0 PL=0
MOVL C00825 V=800.0 PL=0
MOVL C00826 V=800.0 PL=0
MOVL C00827 V=800.0 PL=0
MOVL C00828 V=800.0 PL=0
MOVL C00829 V=800.0 PL=0
MOVL C00830 V=800.0 PL=0
MOVL C00831 V=800.0 PL=0
MOVL C00832 V=800.0 PL=0
MOVL C00833 V=800.0 PL=0
MOVL C00834 V=800.0 PL=0
MOVL C00835 V=800.0 PL=0
MOVL C00836 V=800.0 PL=0
MOVL C00837 V=800.0 PL=0
MOVL C00838 V=800.0 PL=0
MOVL C00839 V=800.0 PL=0
MOVL C00840 V=800.0 PL=0
MOVL C00841 V=800.0 PL=0
MOVL C00842 V=800.0 PL=0
MOVL C00843 V=800.0 PL=0
MOVL C00844 V=800.0 PL=0
MOVL C00845 V=800.0 PL=0
MOVL C00846 V=800.0 PL=0
MOVL C00847 V=800.0 PL=0
MOVL C00848 V=800.0 PL=0
MOVL C00849 V=800.0 PL=0
MOVL C00850 V=800.0 PL=0
MOVL C00851 V=800.0 PL=0
MOVL C00852 V=800.0 PL=0
MOVL C00853 V=800.0 PL=0
MOVL C00854 V=800.0 PL=0
MOVL C00855 V=800.0 PL=0
MOVL C00856 V=800.0 PL=0
MOVL C00857 V=800.0 PL=0
MOVL C00858 V=800.0 PL=0
MOVL C00859 V=800.0 PL=0
MOVL C00860 V=800.0 PL=0
MOVL C00861 V=800.0 PL=0
MOVL C00862 V=800.0 PL=0
MOVL C00863 V=800.0 PL=0
MOVL C00864 V=800.0 PL=0
MOVL C00865 V=800.0 PL=0
MOVL C00866 V=800.0 PL=0
MOVL C00867 V=800.0 PL=0
MOVL C00868 V=800.0 PL=0
MOVL C00869 V=800.0 PL=0
MOVL C00870 V=800.0 PL=0
MOVL C00871 V=800.0 PL=0
MOVL C00872 V=800.0 PL=0
MOVL C00873 V=800.0 PL=0
MOVL C00874 V=800.0 PL=0
MOVL C00875 V=800.0 PL=0
MOVL C00876 V=800.0 PL=0
MOVL C00877 V=800.0 PL=0
MOVL C00878 V=800.0 PL=0
MOVL C00879 V=800.0 PL=0
MOVL C00880 V=800.0 PL=0
MOVL C00881 V=800.0 PL=0
MOVL C00882 V=800.0 PL=0
MOVL C00883 V=800.0 PL=0
MOVL C00884 V=800.0 PL=0
MOVL C00885 V=800.0 PL=0
MOVL C00886 V=800.0 PL=0
MOVL C00887 V=800.0 PL=0
MOVL C00888 V=800.0 PL=0
MOVL C00889 V=800.0 PL=0
MOVL C00890 V=800.0 PL=0
MOVL C00891 V=800.0 PL=0
MOVL C00892 V=800.0 PL=0
MOVL C00893 V=800.0 PL=0
MOVL C00894 V=800.0 PL=0
MOVL C00895 V=800.0 PL=0
MOVL C00896 V=800.0 PL=0
MOVL C00897 V=800.0 PL=0
MOVL C00898 V=800.0 PL=0
MOVL C00899 V=800.0 PL=0
MOVL C00900 V=800.0 PL=0
MOVL C00901 V=800.0 PL=0
MOVL C00902 V=800.0 PL=0
MOVL C00903 V=800.0 PL=0
MOVL C00904 V=800.0 PL=0
MOVL C00905 V=800.0 PL=0
MOVL C00906 V=800.0 PL=0
MOVL C00907 V=800.0 PL=0
MOVL C00908 V=800.0 PL=0
MOVL C00909 V=800.0 PL=0
MOVL C00910 V=800.0 PL=0
MOVL C00911 V=800.0 PL=0
MOVL C00912 V=800.0 PL=0
MOVL C00913 V=800.0 PL=0
MOVL C00914 V=800.0 PL=0
MOVL C00915 V=800.0 PL=0
MOVL C00916 V=800.0 PL=0
MOVL C00917 V=800.0 PL=0
MOVL C00918 V=800.0 PL=0
MOVL C00919 V=800.0 PL=0
MOVL C00920 V=800.0 PL=0
MOVL C00921 V=800.0 PL=0
MOVL C00922 V=800.0 PL=0
MOVL C00923 V=800.0 PL=0
MOVL C00924 V=800.0 PL=0
MOVL C00925 V=800.0 PL=0
MOVL C00926 V=800.0 PL=0
MOVL C00927 V=800.0 PL=0
MOVL C00928 V=800.0 PL=0
MOVL C00929 V=800.0 PL=0
MOVL C00930 V=800.0 PL=0
MOVL C00931 V=800.0 PL=0
MOVL C00932 V=800.0 PL=0
MOVL C00933 V=800.0 PL=0
MOVL C00934 V=800.0 PL=0
MOVL C00935 V=800.0 PL=0
MOVL C00936 V=800.0 PL=0
MOVL C00937 V=800.0 PL=0
MOVL C00938 V=800.0 PL=0
MOVL C00939 V=800.0 PL=0
MOVL C00940 V=800.0 PL=0
MOVL C00941 V=800.0 PL=0
MOVL C00942 V=800.0 PL=0
MOVL C00943 V=800.0 PL=0
MOVL C00944 V=800.0 PL=0
MOVL C00945 V=800.0 PL=0
MOVL C00946 V=800.0 PL=0
MOVL C00947 V=800.0 PL=0
MOVL C00948 V=800.0 PL=0
MOVL C00949 V=800.0 PL=0
MOVL C00950 V=800.0 PL=0
MOVL C00951 V=800.0 PL=0
MOVL C00952 V=800.0 PL=0
MOVL C00953 V=800.0 PL=0
MOVL C00954 V=800.0 PL=0
MOVL C00955 V=800.0 PL=0
MOVL C00956 V=800.0 PL=0
MOVL C00957 V=800.0 PL=0
MOVL C00958 V=800.0 PL=0
MOVL C00959 V=800.0 PL=0
MOVL C00960 V=800.0 PL=0
MOVL C00961 V=800.0 PL=0
MOVL C00962 V=800.0 PL=0
MOVL C00963 V=800.0 PL=0
MOVL C00964 V=800.0 PL=0
MOVL C00965 V=800.0 PL=0
MOVL C00966 V=800.0 PL=0
MOVL C00967 V=800.0 PL=0
MOVL C00968 V=800.0 PL=0
MOVL C00969 V=800.0 PL=0
MOVL C00970 V=800.0 PL=0
MOVL C00971 V=800.0 PL=0
MOVL C00972 V=800.0 PL=0
MOVL C00973 V=800.0 PL=0
MOVL C00974 V=800.0 PL=0
MOVL C00975 V=800.0 PL=0
MOVL C00976 V=800.0 PL=0
MOVL C00977 V=800.0 PL=0
MOVL C00978 V=800.0 PL=0
MOVL C00979 V=800.0 PL=0
MOVL C00980 V=800.0 PL=0
MOVL C00981 V=800.0 PL=0
MOVL C00982 V=800.0 PL=0
MOVL C00983 V=800.0 PL=0
MOVL C00984 V=800.0 PL=0
MOVL C00985 V=800.0 PL=0
MOVL C00986 V=800.0 PL=0
MOVL C00987 V=800.0 PL=0
MOVL C00988 V=800.0 PL=0
MOVL C00989 V=800.0 PL=0
MOVL C00990 V=800.0 PL=0
MOVL C00991 V=800.0 PL=0
MOVL C00992 V=800.0 PL=0
MOVL C00993 V=800.0 PL=0
MOVL C00994 V=800.0 PL=0
MOVL C00995 V=800.0 PL=0
MOVL C00996 V=800.0 PL=0
MOVL C00997 V=800.0 PL=0
MOVL C00998 V=800.0 PL=0
MOVL C00999 V=800.0 PL=0
MOVL C01000 V=800.0 PL=0
MOVL C01001 V=800.0 PL=0
MOVL C01002 V=800.0 PL=0
MOVL C01003 V=800.0 PL=0
MOVL C01004 V=800.0 PL=0
MOVL C01005 V=800.0 PL=0
MOVL C01006 V=800.0 PL=0
MOVL C01007 V=800.0 PL=0
MOVL C01008 V=800.0 PL=0
MOVL C01009 V=800.0 PL=0
MOVL C01010 V=800.0 PL=0
MOVL C01011 V=800.0 PL=0
MOVL C01012 V=800.0 PL=0
MOVL C01013 V=800.0 PL=0
MOVL C01014 V=800.0 PL=0
MOVL C01015 V=800.0 PL=0
MOVL C01016 V=800.0 PL=0
MOVL C01017 V=800.0 PL=0
MOVL C01018 V=800.0 PL=0
MOVL C01019 V=800.0 PL=0
MOVL C01020 V=800.0 PL=0
MOVL C01021 V=800.0 PL=0
MOVL C01022 V=800.0 PL=0
MOVL C01023 V=800.0 PL=0
MOVL C01024 V=800.0 PL=0
MOVL C01025 V=800.0 PL=0
MOVL C01026 V=800.0 PL=0
MOVL C01027 V=800.0 PL=0
MOVL C01028 V=800.0 PL=0
MOVL C01029 V=800.0 PL=0
MOVL C01030 V=800.0 PL=0
MOVL C01031 V=800.0 PL=0
MOVL C01032 V=800.0 PL=0
MOVL C01033 V=800.0 PL=0
MOVL C01034 V=800.0 PL=0
MOVL C01035 V=800.0 PL=0
MOVL C01036 V=800.0 PL=0
MOVL C01037 V=800.0 PL=0
MOVL C01038 V=800.0 PL=0
MOVL C01039 V=800.0 PL=0
MOVL C01040 V=800.0 PL=0
MOVL C01041 V=800.0 PL=0
MOVL C01042 V=800.0 PL=0
MOVL C01043 V=800.0 PL=0
MOVL C01044 V=800.0 PL=0
MOVL C01045 V=800.0 PL=0
MOVL C01046 V=800.0 PL=0
MOVL C01047 V=800.0 PL=0
MOVL C01048 V=800.0 PL=0
MOVL C01049 V=800.0 PL=0
MOVL C01050 V=800.0 PL=0
MOVL C01051 V=800.0 PL=0
MOVL C01052 V=800.0 PL=0
MOVL C01053 V=800.0 PL=0
MOVL C01054 V=800.0 PL=0
MOVL C01055 V=800.0 PL=0
MOVL C01056 V=800.0 PL=0
MOVL C01057 V=800.0 PL=0
MOVL C01058 V=800.0 PL=0
MOVL C01059 V=800.0 PL=0
MOVL C01060 V=800.0 PL=0
MOVL C01061 V=800.0 PL=0
MOVL C01062 V=800.0 PL=0
MOVL C01063 V=800.0 PL=0
MOVL C01064 V=800.0 PL=0
MOVL C01065 V=800.0 PL=0
MOVL C01066 V=800.0 PL=0
MOVL C01067 V=800.0 PL=0
MOVL C01068 V=800.0 PL=0
MOVL C01069 V=800.0 PL=0
MOVL C01070 V=800.0 PL=0
MOVL C01071 V=800.0 PL=0
MOVL C01072 V=800.0 PL=0
MOVL C01073 V=800.0 PL=0
MOVL C01074 V=800.0 PL=0
MOVL C01075 V=800.0 PL=0
MOVL C01076 V=800.0 PL=0
MOVL C01077 V=800.0 PL=0
MOVL C01078 V=800.0 PL=0
MOVL C01079 V=800.0 PL=0
MOVL C01080 V=800.0 PL=0
MOVL C01081 V=800.0 PL=0
MOVL C01082 V=800.0 PL=0
MOVL C01083 V=800.0 PL=0
MOVL C01084 V=800.0 PL=0
MOVL C01085 V=800.0 PL=0
MOVL C01086 V=800.0 PL=0
MOVL C01087 V=800.0 PL=0
MOVL C01088 V=800.0 PL=0
MOVL C01089 V=800.0 PL=0
MOVL C01090 V=800.0 PL=0
MOVL C01091 V=800.0 PL=0
MOVL C01092 V=800.0 PL=0
MOVL C01093 V=800.0 PL=0
MOVL C01094 V=800.0 PL=0
MOVL C01095 V=800.0 PL=0
MOVL C01096 V=800.0 PL=0
MOVL C01097 V=800.0 PL=0
MOVL C01098 V=800.0 PL=0
MOVL C01099 V=800.0 PL=0
MOVL C01100 V=800.0 PL=0
MOVL C01101 V=800.0 PL=0
MOVL C01102 V=800.0 PL=0
MOVL C01103 V=800.0 PL=0
MOVL C01104 V=800.0 PL=0
MOVL C01105 V=800.0 PL=0
MOVL C01106 V=800.0 PL=0
MOVL C01107 V=800.0 PL=0
MOVL C01108 V=800.0 PL=0
MOVL C01109 V=800.0 PL=0
MOVL C01110 V=800.0 PL=0
MOVL C01111 V=800.0 PL=0
MOVL C01112 V=800.0 PL=0
MOVL C01113 V=800.0 PL=0
MOVL C01114 V=800.0 PL=0
MOVL C01115 V=800.0 PL=0
MOVL C01116 V=800.0 PL=0
MOVL C01117 V=800.0 PL=0
MOVL C01118 V=800.0 PL=0
MOVL C01119 V=800.0 PL=0
MOVL C01120 V=800.0 PL=0
MOVL C01121 V=800.0 PL=0
MOVL C01122 V=800.0 PL=0
MOVL C01123 V=800.0 PL=0
MOVL C01124 V=800.0 PL=0
MOVL C01125 V=800.0 PL=0
MOVL C01126 V=800.0 PL=0
MOVL C01127 V=800.0 PL=0
MOVL C01128 V=800.0 PL=0
MOVL C01129 V=800.0 PL=0
MOVL C01130 V=800.0 PL=0
MOVL C01131 V=800.0 PL=0
MOVL C01132 V=800.0 PL=0
MOVL C01133 V=800.0 PL=0
MOVL C01134 V=800.0 PL=0
MOVL C01135 V=800.0 PL=0
MOVL C01136 V=800.0 PL=0
MOVL C01137 V=800.0 PL=0
MOVL C01138 V=800.0 PL=0
MOVL C01139 V=800.0 PL=0
MOVL C01140 V=800.0 PL=0
MOVL C01141 V=800.0 PL=0
MOVL C01142 V=800.0 PL=0
MOVL C01143 V=800.0 PL=0
MOVL C01144 V=800.0 PL=0
MOVL C01145 V=800.0 PL=0
MOVL C01146 V=800.0 PL=0
MOVL C01147 V=800.0 PL=0
MOVL C01148 V=800.0 PL=0
MOVL C01149 V=800.0 PL=0
MOVL C01150 V=800.0 PL=0
MOVL C01151 V=800.0 PL=0
MOVL C01152 V=800.0 PL=0
MOVL C01153 V=800.0 PL=0
MOVL C01154 V=800.0 PL=0
MOVL C01155 V=800.0 PL=0
MOVL C01156 V=800.0 PL=0
MOVL C01157 V=800.0 PL=0
MOVL C01158 V=800.0 PL=0
MOVL C01159 V=800.0 PL=0
MOVL C01160 V=800.0 PL=0
MOVL C01161 V=800.0 PL=0
MOVL C01162 V=800.0 PL=0
MOVL C01163 V=800.0 PL=0
MOVL C01164 V=800.0 PL=0
MOVL C01165 V=800.0 PL=0
MOVL C01166 V=800.0 PL=0
MOVL C01167 V=800.0 PL=0
MOVL C01168 V=800.0 PL=0
MOVL C01169 V=800.0 PL=0
MOVL C01170 V=800.0 PL=0
MOVL C01171 V=800.0 PL=0
MOVL C01172 V=800.0 PL=0
MOVL C01173 V=800.0 PL=0
MOVL C01174 V=800.0 PL=0
MOVL C01175 V=800.0 PL=0
MOVL C01176 V=800.0 PL=0
MOVL C01177 V=800.0 PL=0
MOVL C01178 V=800.0 PL=0
MOVL C01179 V=800.0 PL=0
MOVL C01180 V=800.0 PL=0
MOVL C01181 V=800.0 PL=0
MOVL C01182 V=800.0 PL=0
MOVL C01183 V=800.0 PL=0
MOVL C01184 V=800.0 PL=0
MOVL C01185 V=800.0 PL=0
MOVL C01186 V=800.0 PL=0
MOVL C01187 V=800.0 PL=0
MOVL C01188 V=800.0 PL=0
MOVL C01189 V=800.0 PL=0
MOVL C01190 V=800.0 PL=0
MOVL C01191 V=800.0 PL=0
MOVL C01192 V=800.0 PL=0
MOVL C01193 V=800.0 PL=0
MOVL C01194 V=800.0 PL=0
MOVL C01195 V=800.0 PL=0
MOVL C01196 V=800.0 PL=0
MOVL C01197 V=800.0 PL=0
MOVL C01198 V=800.0 PL=0
MOVL C01199 V=800.0 PL=0
MOVL C01200 V=800.0 PL=0
MOVL C01201 V=800.0 PL=0
MOVL C01202 V=800.0 PL=0
MOVL C01203 V=800.0 PL=0
MOVL C01204 V=800.0 PL=0
MOVL C01205 V=800.0 PL=0
MOVL C01206 V=800.0 PL=0
MOVL C01207 V=800.0 PL=0
MOVL C01208 V=800.0 PL=0
MOVL C01209 V=800.0 PL=0
MOVL C01210 V=800.0 PL=0
MOVL C01211 V=800.0 PL=0
MOVL C01212 V=800.0 PL=0
MOVL C01213 V=800.0 PL=0
MOVL C01214 V=800.0 PL=0
MOVL C01215 V=800.0 PL=0
MOVL C01216 V=800.0 PL=0
MOVL C01217 V=800.0 PL=0
MOVL C01218 V=800.0 PL=0
MOVL C01219 V=800.0 PL=0
MOVL C01220 V=800.0 PL=0
MOVL C01221 V=800.0 PL=0
MOVL C01222 V=800.0 PL=0
MOVL C01223 V=800.0 PL=0
MOVL C01224 V=800.0 PL=0
MOVL C01225 V=800.0 PL=0
MOVL C01226 V=800.0 PL=0
MOVL C01227 V=800.0 PL=0
MOVL C01228 V=800.0 PL=0
MOVL C01229 V=800.0 PL=0
MOVL C01230 V=800.0 PL=0
MOVL C01231 V=800.0 PL=0
MOVL C01232 V=800.0 PL=0
MOVL C01233 V=800.0 PL=0
MOVL C01234 V=800.0 PL=0
MOVL C01235 V=800.0 PL=0
MOVL C01236 V=800.0 PL=0
MOVL C01237 V=800.0 PL=0
MOVL C01238 V=800.0 PL=0
MOVL C01239 V=800.0 PL=0
MOVL C01240 V=800.0 PL=0
MOVL C01241 V=800.0 PL=0
MOVL C01242 V=800.0 PL=0
MOVL C01243 V=800.0 PL=0
MOVL C01244 V=800.0 PL=0
MOVL C01245 V=800.0 PL=0
MOVL C01246 V=800.0 PL=0
MOVL C01247 V=800.0 PL=0
MOVL C01248 V=800.0 PL=0
MOVL C01249 V=800.0 PL=0
MOVL C01250 V=800.0 PL=0
MOVL C01251 V=800.0 PL=0
MOVL C01252 V=800.0 PL=0
MOVL C01253 V=800.0 PL=0
MOVL C01254 V=800.0 PL=0
MOVL C01255 V=800.0 PL=0
MOVL C01256 V=800.0 PL=0
MOVL C01257 V=800.0 PL=0
MOVL C01258 V=800.0 PL=0
MOVL C01259 V=800.0 PL=0
MOVL C01260 V=800.0 PL=0
MOVL C01261 V=800.0 PL=0
MOVL C01262 V=800.0 PL=0
MOVL C01263 V=800.0 PL=0
MOVL C01264 V=800.0 PL=0
MOVL C01265 V=800.0 PL=0
MOVL C01266 V=800.0 PL=0
MOVL C01267 V=800.0 PL=0
MOVL C01268 V=800.0 PL=0
MOVL C01269 V=800.0 PL=0
MOVL C01270 V=800.0 PL=0
MOVL C01271 V=800.0 PL=0
MOVL C01272 V=800.0 PL=0
MOVL C01273 V=800.0 PL=0
MOVL C01274 V=800.0 PL=0
MOVL C01275 V=800.0 PL=0
MOVL C01276 V=800.0 PL=0
MOVL C01277 V=800.0 PL=0
MOVL C01278 V=800.0 PL=0
MOVL C01279 V=800.0 PL=0
MOVL C01280 V=800.0 PL=0
MOVL C01281 V=800.0 PL=0
MOVL C01282 V=800.0 PL=0
MOVL C01283 V=800.0 PL=0
MOVL C01284 V=800.0 PL=0
MOVL C01285 V=800.0 PL=0
MOVL C01286 V=800.0 PL=0
MOVL C01287 V=800.0 PL=0
MOVL C01288 V=800.0 PL=0
MOVL C01289 V=800.0 PL=0
MOVL C01290 V=800.0 PL=0
MOVL C01291 V=800.0 PL=0
MOVL C01292 V=800.0 PL=0
MOVL C01293 V=800.0 PL=0
MOVL C01294 V=800.0 PL=0
MOVL C01295 V=800.0 PL=0
MOVL C01296 V=800.0 PL=0
MOVL C01297 V=800.0 PL=0
MOVL C01298 V=800.0 PL=0
MOVL C01299 V=800.0 PL=0
MOVL C01300 V=800.0 PL=0
MOVL C01301 V=800.0 PL=0
MOVL C01302 V=800.0 PL=0
MOVL C01303 V=800.0 PL=0
MOVL C01304 V=800.0 PL=0
MOVL C01305 V=800.0 PL=0
MOVL C01306 V=800.0 PL=0
MOVL C01307 V=800.0 PL=0
MOVL C01308 V=800.0 PL=0
MOVL C01309 V=800.0 PL=0
MOVL C01310 V=800.0 PL=0
MOVL C01311 V=800.0 PL=0
MOVL C01312 V=800.0 PL=0
MOVL C01313 V=800.0 PL=0
MOVL C01314 V=800.0 PL=0
MOVL C01315 V=800.0 PL=0
MOVL C01316 V=800.0 PL=0
MOVL C01317 V=800.0 PL=0
MOVL C01318 V=800.0 PL=0
MOVL C01319 V=800.0 PL=0
MOVL C01320 V=800.0 PL=0
MOVL C01321 V=800.0 PL=0
MOVL C01322 V=800.0 PL=0
MOVL C01323 V=800.0 PL=0
MOVL C01324 V=800.0 PL=0
MOVL C01325 V=800.0 PL=0
MOVL C01326 V=800.0 PL=0
MOVL C01327 V=800.0 PL=0
MOVL C01328 V=800.0 PL=0
MOVL C01329 V=800.0 PL=0
MOVL C01330 V=800.0 PL=0
MOVL C01331 V=800.0 PL=0
MOVL C01332 V=800.0 PL=0
MOVL C01333 V=800.0 PL=0
MOVL C01334 V=800.0 PL=0
MOVL C01335 V=800.0 PL=0
MOVL C01336 V=800.0 PL=0
MOVL C01337 V=800.0 PL=0
MOVL C01338 V=800.0 PL=0
MOVL C01339 V=800.0 PL=0
MOVL C01340 V=800.0 PL=0
MOVL C01341 V=800.0 PL=0
MOVL C01342 V=800.0 PL=0
MOVL C01343 V=800.0 PL=0
MOVL C01344 V=800.0 PL=0
MOVL C01345 V=800.0 PL=0
MOVL C01346 V=800.0 PL=0
MOVL C01347 V=800.0 PL=0
MOVL C01348 V=800.0 PL=0
MOVL C01349 V=800.0 PL=0
MOVL C01350 V=800.0 PL=0
MOVL C01351 V=800.0 PL=0
MOVL C01352 V=800.0 PL=0
MOVL C01353 V=800.0 PL=0
MOVL C01354 V=800.0 PL=0
MOVL C01355 V=800.0 PL=0
MOVL C01356 V=800.0 PL=0
MOVL C01357 V=800.0 PL=0
MOVL C01358 V=800.0 PL=0
MOVL C01359 V=800.0 PL=0
MOVL C01360 V=800.0 PL=0
MOVL C01361 V=800.0 PL=0
MOVL C01362 V=800.0 PL=0
MOVL C01363 V=800.0 PL=0
MOVL C01364 V=800.0 PL=0
MOVL C01365 V=800.0 PL=0
MOVL C01366 V=800.0 PL=0
MOVL C01367 V=800.0 PL=0
MOVL C01368 V=800.0 PL=0
MOVL C01369 V=800.0 PL=0
MOVL C01370 V=800.0 PL=0
MOVL C01371 V=800.0 PL=0
MOVL C01372 V=800.0 PL=0
MOVL C01373 V=800.0 PL=0
MOVL C01374 V=800.0 PL=0
MOVL C01375 V=800.0 PL=0
MOVL C01376 V=800.0 PL=0
MOVL C01377 V=800.0 PL=0
MOVL C01378 V=800.0 PL=0
MOVL C01379 V=800.0 PL=0
MOVL C01380 V=800.0 PL=0
MOVL C01381 V=800.0 PL=0
MOVL C01382 V=800.0 PL=0
MOVL C01383 V=800.0 PL=0
MOVL C01384 V=800.0 PL=0
MOVL C01385 V=800.0 PL=0
MOVL C01386 V=800.0 PL=0
MOVL C01387 V=800.0 PL=0
MOVL C01388 V=800.0 PL=0
MOVL C01389 V=800.0 PL=0
MOVL C01390 V=800.0 PL=0
MOVL C01391 V=800.0 PL=0
MOVL C01392 V=800.0 PL=0
MOVL C01393 V=800.0 PL=0
MOVL C01394 V=800.0 PL=0
MOVL C01395 V=800.0 PL=0
MOVL C01396 V=800.0 PL=0
MOVL C01397 V=800.0 PL=0
MOVL C01398 V=800.0 PL=0
MOVL C01399 V=800.0 PL=0
MOVL C01400 V=800.0 PL=0
MOVL C01401 V=800.0 PL=0
MOVL C01402 V=800.0 PL=0
MOVL C01403 V=800.0 PL=0
MOVL C01404 V=800.0 PL=0
MOVL C01405 V=800.0 PL=0
MOVL C01406 V=800.0 PL=0
MOVL C01407 V=800.0 PL=0
MOVL C01408 V=800.0 PL=0
MOVL C01409 V=800.0 PL=0
MOVL C01410 V=800.0 PL=0
MOVL C01411 V=800.0 PL=0
MOVL C01412 V=800.0 PL=0
MOVL C01413 V=800.0 PL=0
MOVL C01414 V=800.0 PL=0
MOVL C01415 V=800.0 PL=0
MOVL C01416 V=800.0 PL=0
MOVL C01417 V=800.0 PL=0
MOVL C01418 V=800.0 PL=0
MOVL C01419 V=800.0 PL=0
MOVL C01420 V=800.0 PL=0
MOVL C01421 V=800.0 PL=0
MOVL C01422 V=800.0 PL=0
MOVL C01423 V=800.0 PL=0
MOVL C01424 V=800.0 PL=0
MOVL C01425 V=800.0 PL=0
MOVL C01426 V=800.0 PL=0
MOVL C01427 V=800.0 PL=0
MOVL C01428 V=800.0 PL=0
MOVL C01429 V=800.0 PL=0
MOVL C01430 V=800.0 PL=0
MOVL C01431 V=800.0 PL=0
MOVL C01432 V=800.0 PL=0
MOVL C01433 V=800.0 PL=0
MOVL C01434 V=800.0 PL=0
MOVL C01435 V=800.0 PL=0
MOVL C01436 V=800.0 PL=0
MOVL C01437 V=800.0 PL=0
MOVL C01438 V=800.0 PL=0
MOVL C01439 V=800.0 PL=0
MOVL C01440 V=800.0 PL=0
MOVL C01441 V=800.0 PL=0
MOVL C01442 V=800.0 PL=0
MOVL C01443 V=800.0 PL=0
MOVL C01444 V=800.0 PL=0
MOVL C01445 V=800.0 PL=0
MOVL C01446 V=800.0 PL=0
MOVL C01447 V=800.0 PL=0
MOVL C01448 V=800.0 PL=0
MOVL C01449 V=800.0 PL=0
MOVL C01450 V=800.0 PL=0
MOVL C01451 V=800.0 PL=0
MOVL C01452 V=800.0 PL=0
MOVL C01453 V=800.0 PL=0
MOVL C01454 V=800.0 PL=0
MOVL C01455 V=800.0 PL=0
MOVL C01456 V=800.0 PL=0
MOVL C01457 V=800.0 PL=0
MOVL C01458 V=800.0 PL=0
MOVL C01459 V=800.0 PL=0
MOVL C01460 V=800.0 PL=0
MOVL C01461 V=800.0 PL=0
MOVL C01462 V=800.0 PL=0
MOVL C01463 V=800.0 PL=0
MOVL C01464 V=800.0 PL=0
MOVL C01465 V=800.0 PL=0
MOVL C01466 V=800.0 PL=0
MOVL C01467 V=800.0 PL=0
MOVL C01468 V=800.0 PL=0
MOVL C01469 V=800.0 PL=0
MOVL C01470 V=800.0 PL=0
MOVL C01471 V=800.0 PL=0
MOVL C01472 V=800.0 PL=0
MOVL C01473 V=800.0 PL=0
MOVL C01474 V=800.0 PL=0
MOVL C01475 V=800.0 PL=0
MOVL C01476 V=800.0 PL=0
MOVL C01477 V=800.0 PL=0
MOVL C01478 V=800.0 PL=0
MOVL C01479 V=800.0 PL=0
MOVL C01480 V=800.0 PL=0
MOVL C01481 V=800.0 PL=0
MOVL C01482 V=800.0 PL=0
MOVL C01483 V=800.0 PL=0
MOVL C01484 V=800.0 PL=0
MOVL C01485 V=800.0 PL=0
MOVL C01486 V=800.0 PL=0
MOVL C01487 V=800.0 PL=0
MOVL C01488 V=800.0 PL=0
MOVL C01489 V=800.0 PL=0
MOVL C01490 V=800.0 PL=0
MOVL C01491 V=800.0 PL=0
MOVL C01492 V=800.0 PL=0
MOVL C01493 V=800.0 PL=0
MOVL C01494 V=800.0 PL=0
MOVL C01495 V=800.0 PL=0
MOVL C01496 V=800.0 PL=0
MOVL C01497 V=800.0 PL=0
MOVL C01498 V=800.0 PL=0
MOVL C01499 V=800.0 PL=0
MOVL C01500 V=800.0 PL=0
MOVL C01501 V=800.0 PL=0
MOVL C01502 V=800.0 PL=0
MOVL C01503 V=800.0 PL=0
MOVL C01504 V=800.0 PL=0
MOVL C01505 V=800.0 PL=0
MOVL C01506 V=800.0 PL=0
MOVL C01507 V=800.0 PL=0
MOVL C01508 V=800.0 PL=0
MOVL C01509 V=800.0 PL=0
MOVL C01510 V=800.0 PL=0
MOVL C01511 V=800.0 PL=0
MOVL C01512 V=800.0 PL=0
MOVL C01513 V=800.0 PL=0
MOVL C01514 V=800.0 PL=0
MOVL C01515 V=800.0 PL=0
MOVL C01516 V=800.0 PL=0
MOVL C01517 V=800.0 PL=0
MOVL C01518 V=800.0 PL=0
MOVL C01519 V=800.0 PL=0
MOVL C01520 V=800.0 PL=0
MOVL C01521 V=800.0 PL=0
MOVL C01522 V=800.0 PL=0
MOVL C01523 V=800.0 PL=0
MOVL C01524 V=800.0 PL=0
MOVL C01525 V=800.0 PL=0
MOVL C01526 V=800.0 PL=0
MOVL C01527 V=800.0 PL=0
MOVL C01528 V=800.0 PL=0
MOVL C01529 V=800.0 PL=0
MOVL C01530 V=800.0 PL=0
MOVL C01531 V=800.0 PL=0
MOVL C01532 V=800.0 PL=0
MOVL C01533 V=800.0 PL=0
MOVL C01534 V=800.0 PL=0
MOVL C01535 V=800.0 PL=0
MOVL C01536 V=800.0 PL=0
MOVL C01537 V=800.0 PL=0
MOVL C01538 V=800.0 PL=0
MOVL C01539 V=800.0 PL=0
MOVL C01540 V=800.0 PL=0
MOVL C01541 V=800.0 PL=0
MOVL C01542 V=800.0 PL=0
MOVL C01543 V=800.0 PL=0
MOVL C01544 V=800.0 PL=0
MOVL C01545 V=800.0 PL=0
MOVL C01546 V=800.0 PL=0
MOVL C01547 V=800.0 PL=0
MOVL C01548 V=800.0 PL=0
MOVL C01549 V=800.0 PL=0
MOVL C01550 V=800.0 PL=0
MOVL C01551 V=800.0 PL=0
MOVL C01552 V=800.0 PL=0
MOVL C01553 V=800.0 PL=0
MOVL C01554 V=800.0 PL=0
MOVL C01555 V=800.0 PL=0
MOVL C01556 V=800.0 PL=0
MOVL C01557 V=800.0 PL=0
MOVL C01558 V=800.0 PL=0
MOVL C01559 V=800.0 PL=0
MOVL C01560 V=800.0 PL=0
MOVL C01561 V=800.0 PL=0
MOVL C01562 V=800.0 PL=0
MOVL C01563 V=800.0 PL=0
MOVL C01564 V=800.0 PL=0
MOVL C01565 V=800.0 PL=0
MOVL C01566 V=800.0 PL=0
MOVL C01567 V=800.0 PL=0
MOVL C01568 V=800.0 PL=0
MOVL C01569 V=800.0 PL=0
MOVL C01570 V=800.0 PL=0
MOVL C01571 V=800.0 PL=0
MOVL C01572 V=800.0 PL=0
MOVL C01573 V=800.0 PL=0
MOVL C01574 V=800.0 PL=0
MOVL C01575 V=800.0 PL=0
MOVL C01576 V=800.0 PL=0
MOVL C01577 V=800.0 PL=0
MOVL C01578 V=800.0 PL=0
MOVL C01579 V=800.0 PL=0
MOVL C01580 V=800.0 PL=0
MOVL C01581 V=800.0 PL=0
MOVL C01582 V=800.0 PL=0
MOVL C01583 V=800.0 PL=0
MOVL C01584 V=800.0 PL=0
MOVL C01585 V=800.0 PL=0
MOVL C01586 V=800.0 PL=0
MOVL C01587 V=800.0 PL=0
MOVL C01588 V=800.0 PL=0
MOVL C01589 V=800.0 PL=0
MOVL C01590 V=800.0 PL=0
MOVL C01591 V=800.0 PL=0
MOVL C01592 V=800.0 PL=0
MOVL C01593 V=800.0 PL=0
MOVL C01594 V=800.0 PL=0
MOVL C01595 V=800.0 PL=0
MOVL C01596 V=800.0 PL=0
MOVL C01597 V=800.0 PL=0
MOVL C01598 V=800.0 PL=0
MOVL C01599 V=800.0 PL=0
MOVL C01600 V=800.0 PL=0
MOVL C01601 V=800.0 PL=0
MOVL C01602 V=800.0 PL=0
MOVL C01603 V=800.0 PL=0
MOVL C01604 V=800.0 PL=0
MOVL C01605 V=800.0 PL=0
MOVL C01606 V=800.0 PL=0
MOVL C01607 V=800.0 PL=0
MOVL C01608 V=800.0 PL=0
MOVL C01609 V=800.0 PL=0
MOVL C01610 V=800.0 PL=0
MOVL C01611 V=800.0 PL=0
MOVL C01612 V=800.0 PL=0
MOVL C01613 V=800.0 PL=0
MOVL C01614 V=800.0 PL=0
MOVL C01615 V=800.0 PL=0
MOVL C01616 V=800.0 PL=0
MOVL C01617 V=800.0 PL=0
MOVL C01618 V=800.0 PL=0
MOVL C01619 V=800.0 PL=0
MOVL C01620 V=800.0 PL=0
MOVL C01621 V=800.0 PL=0
MOVL C01622 V=800.0 PL=0
MOVL C01623 V=800.0 PL=0
MOVL C01624 V=800.0 PL=0
MOVL C01625 V=800.0 PL=0
MOVL C01626 V=800.0 PL=0
MOVL C01627 V=800.0 PL=0
MOVL C01628 V=800.0 PL=0
MOVL C01629 V=800.0 PL=0
MOVL C01630 V=800.0 PL=0
MOVL C01631 V=800.0 PL=0
MOVL C01632 V=800.0 PL=0
MOVL C01633 V=800.0 PL=0
MOVL C01634 V=800.0 PL=0
MOVL C01635 V=800.0 PL=0
MOVL C01636 V=800.0 PL=0
MOVL C01637 V=800.0 PL=0
MOVL C01638 V=800.0 PL=0
MOVL C01639 V=800.0 PL=0
MOVL C01640 V=800.0 PL=0
MOVL C01641 V=800.0 PL=0
MOVL C01642 V=800.0 PL=0
MOVL C01643 V=800.0 PL=0
MOVL C01644 V=800.0 PL=0
MOVL C01645 V=800.0 PL=0
MOVL C01646 V=800.0 PL=0
MOVL C01647 V=800.0 PL=0
MOVL C01648 V=800.0 PL=0
MOVL C01649 V=800.0 PL=0
MOVL C01650 V=800.0 PL=0
MOVL C01651 V=800.0 PL=0
MOVL C01652 V=800.0 PL=0
MOVL C01653 V=800.0 PL=0
MOVL C01654 V=800.0 PL=0
MOVL C01655 V=800.0 PL=0
MOVL C01656 V=800.0 PL=0
MOVL C01657 V=800.0 PL=0
MOVL C01658 V=800.0 PL=0
MOVL C01659 V=800.0 PL=0
MOVL C01660 V=800.0 PL=0
MOVL C01661 V=800.0 PL=0
MOVL C01662 V=800.0 PL=0
MOVL C01663 V=800.0 PL=0
MOVL C01664 V=800.0 PL=0
MOVL C01665 V=800.0 PL=0
MOVL C01666 V=800.0 PL=0
MOVL C01667 V=800.0 PL=0
MOVL C01668 V=800.0 PL=0
MOVL C01669 V=800.0 PL=0
MOVL C01670 V=800.0 PL=0
MOVL C01671 V=800.0 PL=0
MOVL C01672 V=800.0 PL=0
MOVL C01673 V=800.0 PL=0
MOVL C01674 V=800.0 PL=0
MOVL C01675 V=800.0 PL=0
MOVL C01676 V=800.0 PL=0
MOVL C01677 V=800.0 PL=0
MOVL C01678 V=800.0 PL=0
MOVL C01679 V=800.0 PL=0
MOVL C01680 V=800.0 PL=0
MOVL C01681 V=800.0 PL=0
MOVL C01682 V=800.0 PL=0
MOVL C01683 V=800.0 PL=0
MOVL C01684 V=800.0 PL=0
MOVL C01685 V=800.0 PL=0
MOVL C01686 V=800.0 PL=0
MOVL C01687 V=800.0 PL=0
MOVL C01688 V=800.0 PL=0
MOVL C01689 V=800.0 PL=0
MOVL C01690 V=800.0 PL=0
MOVL C01691 V=800.0 PL=0
MOVL C01692 V=800.0 PL=0
MOVL C01693 V=800.0 PL=0
MOVL C01694 V=800.0 PL=0
MOVL C01695 V=800.0 PL=0
MOVL C01696 V=800.0 PL=0
MOVL C01697 V=800.0 PL=0
MOVL C01698 V=800.0 PL=0
MOVL C01699 V=800.0 PL=0
MOVL C01700 V=800.0 PL=0
MOVL C01701 V=800.0 PL=0
MOVL C01702 V=800.0 PL=0
MOVL C01703 V=800.0 PL=0
MOVL C01704 V=800.0 PL=0
MOVL C01705 V=800.0 PL=0
MOVL C01706 V=800.0 PL=0
MOVL C01707 V=800.0 PL=0
MOVL C01708 V=800.0 PL=0
MOVL C01709 V=800.0 PL=0
MOVL C01710 V=800.0 PL=0
MOVL C01711 V=800.0 PL=0
MOVL C01712 V=800.0 PL=0
MOVL C01713 V=800.0 PL=0
MOVL C01714 V=800.0 PL=0
MOVL C01715 V=800.0 PL=0
MOVL C01716 V=800.0 PL=0
MOVL C01717 V=800.0 PL=0
MOVL C01718 V=800.0 PL=0
MOVL C01719 V=800.0 PL=0
MOVL C01720 V=800.0 PL=0
MOVL C01721 V=800.0 PL=0
MOVL C01722 V=800.0 PL=0
MOVL C01723 V=800.0 PL=0
MOVL C01724 V=800.0 PL=0
MOVL C01725 V=800.0 PL=0
MOVL C01726 V=800.0 PL=0
MOVL C01727 V=800.0 PL=0
MOVL C01728 V=800.0 PL=0
MOVL C01729 V=800.0 PL=0
MOVL C01730 V=800.0 PL=0
MOVL C01731 V=800.0 PL=0
MOVL C01732 V=800.0 PL=0
MOVL C01733 V=800.0 PL=0
MOVL C01734 V=800.0 PL=0
MOVL C01735 V=800.0 PL=0
MOVL C01736 V=800.0 PL=0
MOVL C01737 V=800.0 PL=0
MOVL C01738 V=800.0 PL=0
MOVL C01739 V=800.0 PL=0
MOVL C01740 V=800.0 PL=0
MOVL C01741 V=800.0 PL=0
MOVL C01742 V=800.0 PL=0
MOVL C01743 V=800.0 PL=0
MOVL C01744 V=800.0 PL=0
MOVL C01745 V=800.0 PL=0
MOVL C01746 V=800.0 PL=0
MOVL C01747 V=800.0 PL=0
MOVL C01748 V=800.0 PL=0
MOVL C01749 V=800.0 PL=0
MOVL C01750 V=800.0 PL=0
MOVL C01751 V=800.0 PL=0
MOVL C01752 V=800.0 PL=0
MOVL C01753 V=800.0 PL=0
MOVL C01754 V=800.0 PL=0
MOVL C01755 V=800.0 PL=0
MOVL C01756 V=800.0 PL=0
MOVL C01757 V=800.0 PL=0
MOVL C01758 V=800.0 PL=0
MOVL C01759 V=800.0 PL=0
MOVL C01760 V=800.0 PL=0
MOVL C01761 V=800.0 PL=0
MOVL C01762 V=800.0 PL=0
MOVL C01763 V=800.0 PL=0
MOVL C01764 V=800.0 PL=0
MOVL C01765 V=800.0 PL=0
MOVL C01766 V=800.0 PL=0
MOVL C01767 V=800.0 PL=0
MOVL C01768 V=800.0 PL=0
MOVL C01769 V=800.0 PL=0
MOVL C01770 V=800.0 PL=0
MOVL C01771 V=800.0 PL=0
MOVL C01772 V=800.0 PL=0
MOVL C01773 V=800.0 PL=0
MOVL C01774 V=800.0 PL=0
MOVL C01775 V=800.0 PL=0
MOVL C01776 V=800.0 PL=0
MOVL C01777 V=800.0 PL=0
MOVL C01778 V=800.0 PL=0
MOVL C01779 V=800.0 PL=0
MOVL C01780 V=800.0 PL=0
MOVL C01781 V=800.0 PL=0
MOVL C01782 V=800.0 PL=0
MOVL C01783 V=800.0 PL=0
MOVL C01784 V=800.0 PL=0
MOVL C01785 V=800.0 PL=0
MOVL C01786 V=800.0 PL=0
MOVL C01787 V=800.0 PL=0
MOVL C01788 V=800.0 PL=0
MOVL C01789 V=800.0 PL=0
MOVL C01790 V=800.0 PL=0
MOVL C01791 V=800.0 PL=0
MOVL C01792 V=800.0 PL=0
MOVL C01793 V=800.0 PL=0
MOVL C01794 V=800.0 PL=0
MOVL C01795 V=800.0 PL=0
MOVL C01796 V=800.0 PL=0
MOVL C01797 V=800.0 PL=0
MOVL C01798 V=800.0 PL=0
MOVL C01799 V=800.0 PL=0
MOVL C01800 V=800.0 PL=0
MOVL C01801 V=800.0 PL=0
MOVL C01802 V=800.0 PL=0
MOVL C01803 V=800.0 PL=0
MOVL C01804 V=800.0 PL=0
MOVL C01805 V=800.0 PL=0
MOVL C01806 V=800.0 PL=0
MOVL C01807 V=800.0 PL=0
MOVL C01808 V=800.0 PL=0
MOVL C01809 V=800.0 PL=0
MOVL C01810 V=800.0 PL=0
MOVL C01811 V=800.0 PL=0
MOVL C01812 V=800.0 PL=0
MOVL C01813 V=800.0 PL=0
MOVL C01814 V=800.0 PL=0
MOVL C01815 V=800.0 PL=0
MOVL C01816 V=800.0 PL=0
MOVL C01817 V=800.0 PL=0
MOVL C01818 V=800.0 PL=0
MOVL C01819 V=800.0 PL=0
MOVL C01820 V=800.0 PL=0
MOVL C01821 V=800.0 PL=0
MOVL C01822 V=800.0 PL=0
MOVL C01823 V=800.0 PL=0
